LIN {X 0,Y 424.138,Z 935.188,A -85,B 0,C 180,E1 -9807.151,E2 -9807.151} C_VEL
LIN {X 0,Y 424.125,Z 936.443,A -85,B 0,C 180,E1 -9808.101,E2 -9808.101} C_VEL
LIN {X 0,Y 424.085,Z 937.224,A -85,B 0,C 180,E1 -9809.05,E2 -9809.05} C_VEL
LIN {X 0,Y 424.081,Z 937.52,A -85,B 0,C 180,E1 -9810,E2 -9810} C_VEL
LIN {X 0,Y 424.085,Z 937.223,A -85,B 0,C 180,E1 -9810.95,E2 -9810.95} C_VEL
LIN {X 0,Y 424.125,Z 936.441,A -85,B 0,C 180,E1 -9811.899,E2 -9811.899} C_VEL
LIN {X 0,Y 424.138,Z 935.183,A -85,B 0,C 180,E1 -9812.849,E2 -9812.849} C_VEL
LIN {X 0,Y 424.185,Z 932.271,A -85,B 0,C 180,E1 -9814.276,E2 -9814.276} C_VEL
LIN {X 0,Y 424.292,Z 929.619,A -85,B 0,C 180,E1 -9815.227,E2 -9815.227} C_VEL
LIN {X 0,Y 424.459,Z 924.427,A -85,B 0,C 180,E1 -9816.656,E2 -9816.656} C_VEL
LIN {X 0,Y 424.787,Z 917.59,A -85,B 0,C 180,E1 -9818.084,E2 -9818.084} C_VEL
LIN {X 0,Y 425.186,Z 910.116,A -85,B 0,C 180,E1 -9819.274,E2 -9819.274} C_VEL
LIN {X 0,Y 425.577,Z 902.747,A -85,B 0,C 180,E1 -9820.226,E2 -9820.226} C_VEL
LIN {X 0,Y 426.04,Z 894.86,A -85,B 0,C 180,E1 -9821.056,E2 -9821.056} C_VEL
LIN {X 0,Y 426.464,Z 886.526,A -85,B 0,C 180,E1 -9821.767,E2 -9821.767} C_VEL
LIN {X 0,Y 426.955,Z 877.803,A -85,B 0,C 180,E1 -9822.356,E2 -9822.356} C_VEL
LIN {X 0,Y 427.276,Z 865.987,A -85,B 0,C 180,E1 -9822.951,E2 -9822.951} C_VEL
LIN {X 0,Y 427.656,Z 855.955,A -85,B 0,C 180,E1 -9823.271,E2 -9823.271} C_VEL
LIN {X 0,Y 427.862,Z 833.743,A -85,B 0,C 180,E1 -9823.678,E2 -9823.678} C_VEL
LIN {X 0,Y 427.935,Z 796.078,A -85,B 0,C 180,E1 -9824.313,E2 -9824.313} C_VEL
LIN {X 0,Y 425.44,Z 777.594,A -85,B 0,C 180,E1 -9824.737,E2 -9824.737} C_VEL
LIN {X 0,Y 425.535,Z 774.648,A -85,B 0,C 180,E1 -9825.322,E2 -9825.322} C_VEL
LIN {X 0,Y 426.176,Z 760.658,A -85,B 0,C 180,E1 -9828.509,E2 -9828.509} C_VEL
LIN {X 0,Y 427.088,Z 745.503,A -85,B 0,C 180,E1 -9831.985,E2 -9831.985} C_VEL
LIN {X 0,Y 426.388,Z 740.059,A -85,B 0,C 180,E1 -9833.302,E2 -9833.302} C_VEL
LIN {X 0,Y 425.384,Z 734.368,A -85,B 0,C 180,E1 -9834.762,E2 -9834.762} C_VEL
LIN {X 0,Y 425.35,Z 734.312,A -85,B 0,C 180,E1 -9837.558,E2 -9837.558} C_VEL
LIN {X 0,Y 425.288,Z 734.304,A -85,B 0,C 180,E1 -9840.816,E2 -9840.816} C_VEL
LIN {X 0,Y 425.312,Z 734.317,A -85,B 0,C 180,E1 -9844.288,E2 -9844.288} C_VEL
LIN {X 0,Y 425.287,Z 734.323,A -85,B 0,C 180,E1 -9847.693,E2 -9847.693} C_VEL
LIN {X 0,Y 425.286,Z 734.31,A -85,B 0,C 180,E1 -9850.521,E2 -9850.521} C_VEL
LIN {X 0,Y 425.266,Z 734.324,A -85,B 0,C 180,E1 -9853.955,E2 -9853.955} C_VEL
LIN {X 0,Y 425.282,Z 734.317,A -85,B 0,C 180,E1 -9857.348,E2 -9857.348} C_VEL
LIN {X 0,Y 425.308,Z 734.283,A -85,B 0,C 180,E1 -9859.875,E2 -9859.875} C_VEL
LIN {X 0,Y 425.287,Z 734.303,A -85,B 0,C 180,E1 -9862.487,E2 -9862.487} C_VEL
LIN {X 0,Y 425.309,Z 734.32,A -85,B 0,C 180,E1 -9865.818,E2 -9865.818} C_VEL
LIN {X 0,Y 425.291,Z 734.315,A -85,B 0,C 180,E1 -9869.239,E2 -9869.239} C_VEL
LIN {X 0,Y 425.351,Z 734.311,A -85,B 0,C 180,E1 -9872.443,E2 -9872.443} C_VEL
LIN {X 0,Y 425.353,Z 734.312,A -85,B 0,C 180,E1 -9875.602,E2 -9875.602} C_VEL
LIN {X 0,Y 425.295,Z 734.306,A -85,B 0,C 180,E1 -9878.682,E2 -9878.682} C_VEL
LIN {X 0,Y 425.335,Z 734.311,A -85,B 0,C 180,E1 -9881.703,E2 -9881.703} C_VEL
LIN {X 0,Y 425.35,Z 734.308,A -85,B 0,C 180,E1 -9884.671,E2 -9884.671} C_VEL
LIN {X 0,Y 425.414,Z 734.289,A -85,B 0,C 180,E1 -9887.598,E2 -9887.598} C_VEL
LIN {X 0,Y 425.444,Z 734.297,A -85,B 0,C 180,E1 -9891.45,E2 -9891.45} C_VEL
LIN {X 0,Y 425.553,Z 734.289,A -85,B 0,C 180,E1 -9894.313,E2 -9894.313} C_VEL
LIN {X 0,Y 425.575,Z 734.267,A -85,B 0,C 180,E1 -9898.107,E2 -9898.107} C_VEL
LIN {X 0,Y 425.706,Z 734.26,A -85,B 0,C 180,E1 -9900,E2 -9900} C_VEL
LIN {X 0,Y 425.559,Z 734.287,A -85,B 0,C 180,E1 -9902.84,E2 -9902.84} C_VEL
LIN {X 0,Y 425.53,Z 734.277,A -85,B 0,C 180,E1 -9906.639,E2 -9906.639} C_VEL
LIN {X 0,Y 425.402,Z 734.298,A -85,B 0,C 180,E1 -9909.509,E2 -9909.509} C_VEL
LIN {X 0,Y 425.395,Z 734.31,A -85,B 0,C 180,E1 -9912.904,E2 -9912.904} C_VEL
LIN {X 0,Y 425.363,Z 734.301,A -85,B 0,C 180,E1 -9916.605,E2 -9916.605} C_VEL
LIN {X 0,Y 425.33,Z 734.31,A -85,B 0,C 180,E1 -9919.636,E2 -9919.636} C_VEL
LIN {X 0,Y 425.289,Z 734.319,A -85,B 0,C 180,E1 -9922.339,E2 -9922.339} C_VEL
LIN {X 0,Y 425.293,Z 734.307,A -85,B 0,C 180,E1 -9925.446,E2 -9925.446} C_VEL
LIN {X 0,Y 425.35,Z 734.31,A -85,B 0,C 180,E1 -9927.558,E2 -9927.558} C_VEL
LIN {X 0,Y 425.289,Z 734.321,A -85,B 0,C 180,E1 -9930.816,E2 -9930.816} C_VEL
LIN {X 0,Y 425.311,Z 734.309,A -85,B 0,C 180,E1 -9934.288,E2 -9934.288} C_VEL
LIN {X 0,Y 425.28,Z 734.32,A -85,B 0,C 180,E1 -9937.694,E2 -9937.694} C_VEL
LIN {X 0,Y 425.278,Z 734.308,A -85,B 0,C 180,E1 -9940.52,E2 -9940.52} C_VEL
LIN {X 0,Y 425.262,Z 734.307,A -85,B 0,C 180,E1 -9943.956,E2 -9943.956} C_VEL
LIN {X 0,Y 425.275,Z 734.325,A -85,B 0,C 180,E1 -9947.347,E2 -9947.347} C_VEL
LIN {X 0,Y 425.286,Z 734.312,A -85,B 0,C 180,E1 -9949.873,E2 -9949.873} C_VEL
LIN {X 0,Y 425.278,Z 734.311,A -85,B 0,C 180,E1 -9952.489,E2 -9952.489} C_VEL
LIN {X 0,Y 425.307,Z 734.321,A -85,B 0,C 180,E1 -9955.817,E2 -9955.817} C_VEL
LIN {X 0,Y 425.291,Z 734.312,A -85,B 0,C 180,E1 -9959.239,E2 -9959.239} C_VEL
LIN {X 0,Y 425.273,Z 734.322,A -85,B 0,C 180,E1 -9962.437,E2 -9962.437} C_VEL
LIN {X 0,Y 425.347,Z 734.317,A -85,B 0,C 180,E1 -9965.602,E2 -9965.602} C_VEL
LIN {X 0,Y 425.3,Z 734.318,A -85,B 0,C 180,E1 -9968.682,E2 -9968.682} C_VEL
LIN {X 0,Y 425.396,Z 734.425,A -85,B 0,C 180,E1 -9969.783,E2 -9969.783} C_VEL
LIN {X 0,Y 426.02,Z 739.289,A -85,B 0,C 180,E1 -9971.235,E2 -9971.235} C_VEL
LIN {X 0,Y 425.751,Z 748.087,A -85,B 0,C 180,E1 -9973.703,E2 -9973.703} C_VEL
LIN {X 0,Y 425.491,Z 754.134,A -85,B 0,C 180,E1 -9975.297,E2 -9975.297} C_VEL
LIN {X 0,Y 426.166,Z 757.896,A -85,B 0,C 180,E1 -9975.435,E2 -9975.435} C_VEL
LIN {X 0,Y 428.26,Z 770.133,A -85,B 0,C 180,E1 -9975.717,E2 -9975.717} C_VEL
LIN {X 0,Y 427.782,Z 829.524,A -85,B 0,C 180,E1 -9976.733,E2 -9976.733} C_VEL
LIN {X 0,Y 427.629,Z 839.402,A -85,B 0,C 180,E1 -9977.03,E2 -9977.03} C_VEL
LIN {X 0,Y 427.198,Z 850.542,A -85,B 0,C 180,E1 -9977.53,E2 -9977.53} C_VEL
LIN {X 0,Y 426.816,Z 861.387,A -85,B 0,C 180,E1 -9978.243,E2 -9978.243} C_VEL
LIN {X 0,Y 426.333,Z 869.786,A -85,B 0,C 180,E1 -9978.952,E2 -9978.952} C_VEL
LIN {X 0,Y 425.93,Z 877.709,A -85,B 0,C 180,E1 -9979.783,E2 -9979.783} C_VEL
LIN {X 0,Y 425.588,Z 883.399,A -85,B 0,C 180,E1 -9980.495,E2 -9980.495} C_VEL
LIN {X 0,Y 425.435,Z 885.864,A -85,B 0,C 180,E1 -9980.84,E2 -9980.84} C_VEL
LIN {X 0,Y 424.575,Z 889.849,A -85,B 0,C 180,E1 -9981.419,E2 -9981.419} C_VEL
LIN {X 0,Y 421.471,Z 895.791,A -85,B 0,C 180,E1 -9982.412,E2 -9982.412} C_VEL
LIN {X 0,Y 418.358,Z 900.822,A -85,B 0,C 180,E1 -9983.502,E2 -9983.502} C_VEL
LIN {X 0,Y 417.496,Z 903.376,A -85,B 0,C 180,E1 -9984.225,E2 -9984.225} C_VEL
LIN {X 0,Y 417.271,Z 906.303,A -85,B 0,C 180,E1 -9985.169,E2 -9985.169} C_VEL
LIN {X 0,Y 417.217,Z 908.62,A -85,B 0,C 180,E1 -9986.136,E2 -9986.136} C_VEL
LIN {X 0,Y 417.187,Z 910.384,A -85,B 0,C 180,E1 -9987.103,E2 -9987.103} C_VEL
LIN {X 0,Y 417.082,Z 911.659,A -85,B 0,C 180,E1 -9988.069,E2 -9988.069} C_VEL
LIN {X 0,Y 417.012,Z 912.464,A -85,B 0,C 180,E1 -9989.034,E2 -9989.034} C_VEL
LIN {X 0,Y 417.002,Z 912.77,A -85,B 0,C 180,E1 -9990,E2 -9990} C_VEL
LIN {X 0,Y 417.012,Z 912.495,A -85,B 0,C 180,E1 -9990.966,E2 -9990.966} C_VEL
LIN {X 0,Y 417.082,Z 911.751,A -85,B 0,C 180,E1 -9991.931,E2 -9991.931} C_VEL
LIN {X 0,Y 417.186,Z 910.54,A -85,B 0,C 180,E1 -9992.897,E2 -9992.897} C_VEL
LIN {X 0,Y 417.249,Z 907.697,A -85,B 0,C 180,E1 -9994.347,E2 -9994.347} C_VEL
LIN {X 0,Y 417.362,Z 905.108,A -85,B 0,C 180,E1 -9995.314,E2 -9995.314} C_VEL
LIN {X 0,Y 417.689,Z 900.007,A -85,B 0,C 180,E1 -9996.764,E2 -9996.764} C_VEL
LIN {X 0,Y 417.909,Z 894.523,A -85,B 0,C 180,E1 -9997.975,E2 -9997.975} C_VEL
LIN {X 0,Y 418.366,Z 887.629,A -85,B 0,C 180,E1 -9999.183,E2 -9999.183} C_VEL
LIN {X 0,Y 418.886,Z 879.709,A -85,B 0,C 180,E1 -10000.269,E2 -10000.269} C_VEL
LIN {X 0,Y 419.285,Z 872.158,A -85,B 0,C 180,E1 -10001.114,E2 -10001.114} C_VEL
LIN {X 0,Y 419.706,Z 864.241,A -85,B 0,C 180,E1 -10001.837,E2 -10001.837} C_VEL
LIN {X 0,Y 420.074,Z 856.064,A -85,B 0,C 180,E1 -10002.439,E2 -10002.439} C_VEL
LIN {X 0,Y 420.485,Z 847.776,A -85,B 0,C 180,E1 -10002.918,E2 -10002.918} C_VEL
LIN {X 0,Y 420.763,Z 838.827,A -85,B 0,C 180,E1 -10003.308,E2 -10003.308} C_VEL
LIN {X 0,Y 420.914,Z 829.602,A -85,B 0,C 180,E1 -10003.585,E2 -10003.585} C_VEL
LIN {X 0,Y 421.274,Z 770.019,A -85,B 0,C 180,E1 -10004.625,E2 -10004.625} C_VEL
LIN {X 0,Y 418.456,Z 754.177,A -85,B 0,C 180,E1 -10005.027,E2 -10005.027} C_VEL
LIN {X 0,Y 418.992,Z 743.301,A -85,B 0,C 180,E1 -10008.078,E2 -10008.078} C_VEL
LIN {X 0,Y 418.819,Z 738.045,A -85,B 0,C 180,E1 -10009.61,E2 -10009.61} C_VEL
LIN {X 0,Y 418.337,Z 735.274,A -85,B 0,C 180,E1 -10010.501,E2 -10010.501} C_VEL
LIN {X 0,Y 418.274,Z 735.191,A -85,B 0,C 180,E1 -10013.782,E2 -10013.782} C_VEL
LIN {X 0,Y 418.226,Z 735.2,A -85,B 0,C 180,E1 -10017.047,E2 -10017.047} C_VEL
LIN {X 0,Y 418.243,Z 735.198,A -85,B 0,C 180,E1 -10020.272,E2 -10020.272} C_VEL
LIN {X 0,Y 418.249,Z 735.195,A -85,B 0,C 180,E1 -10023.677,E2 -10023.677} C_VEL
LIN {X 0,Y 418.24,Z 735.188,A -85,B 0,C 180,E1 -10027.224,E2 -10027.224} C_VEL
LIN {X 0,Y 418.244,Z 735.185,A -85,B 0,C 180,E1 -10029.683,E2 -10029.683} C_VEL
LIN {X 0,Y 418.231,Z 735.201,A -85,B 0,C 180,E1 -10032.321,E2 -10032.321} C_VEL
LIN {X 0,Y 418.237,Z 735.187,A -85,B 0,C 180,E1 -10035.109,E2 -10035.109} C_VEL
LIN {X 0,Y 418.235,Z 735.163,A -85,B 0,C 180,E1 -10037.766,E2 -10037.766} C_VEL
LIN {X 0,Y 418.25,Z 735.188,A -85,B 0,C 180,E1 -10040.62,E2 -10040.62} C_VEL
LIN {X 0,Y 418.244,Z 735.196,A -85,B 0,C 180,E1 -10043.976,E2 -10043.976} C_VEL
LIN {X 0,Y 418.258,Z 735.191,A -85,B 0,C 180,E1 -10047.156,E2 -10047.156} C_VEL
LIN {X 0,Y 418.27,Z 735.199,A -85,B 0,C 180,E1 -10050.895,E2 -10050.895} C_VEL
LIN {X 0,Y 418.27,Z 735.179,A -85,B 0,C 180,E1 -10054.096,E2 -10054.096} C_VEL
LIN {X 0,Y 418.234,Z 735.202,A -85,B 0,C 180,E1 -10057.263,E2 -10057.263} C_VEL
LIN {X 0,Y 418.285,Z 735.188,A -85,B 0,C 180,E1 -10060.364,E2 -10060.364} C_VEL
LIN {X 0,Y 418.318,Z 735.178,A -85,B 0,C 180,E1 -10063.405,E2 -10063.405} C_VEL
LIN {X 0,Y 418.348,Z 735.185,A -85,B 0,C 180,E1 -10066.999,E2 -10066.999} C_VEL
LIN {X 0,Y 418.342,Z 735.177,A -85,B 0,C 180,E1 -10070.329,E2 -10070.329} C_VEL
LIN {X 0,Y 418.515,Z 735.143,A -85,B 0,C 180,E1 -10072.279,E2 -10072.279} C_VEL
LIN {X 0,Y 418.513,Z 735.155,A -85,B 0,C 180,E1 -10074.217,E2 -10074.217} C_VEL
LIN {X 0,Y 418.547,Z 735.157,A -85,B 0,C 180,E1 -10078.075,E2 -10078.075} C_VEL
LIN {X 0,Y 418.673,Z 735.136,A -85,B 0,C 180,E1 -10080,E2 -10080} C_VEL
LIN {X 0,Y 418.503,Z 735.146,A -85,B 0,C 180,E1 -10082.888,E2 -10082.888} C_VEL
LIN {X 0,Y 418.49,Z 735.164,A -85,B 0,C 180,E1 -10086.751,E2 -10086.751} C_VEL
LIN {X 0,Y 418.343,Z 735.183,A -85,B 0,C 180,E1 -10089.671,E2 -10089.671} C_VEL
LIN {X 0,Y 418.348,Z 735.168,A -85,B 0,C 180,E1 -10093.001,E2 -10093.001} C_VEL
LIN {X 0,Y 418.315,Z 735.186,A -85,B 0,C 180,E1 -10096.736,E2 -10096.736} C_VEL
LIN {X 0,Y 418.301,Z 735.185,A -85,B 0,C 180,E1 -10099.801,E2 -10099.801} C_VEL
LIN {X 0,Y 418.29,Z 735.189,A -85,B 0,C 180,E1 -10103.781,E2 -10103.781} C_VEL
LIN {X 0,Y 418.311,Z 735.185,A -85,B 0,C 180,E1 -10107.07,E2 -10107.07} C_VEL
LIN {X 0,Y 418.245,Z 735.192,A -85,B 0,C 180,E1 -10110.272,E2 -10110.272} C_VEL
LIN {X 0,Y 418.25,Z 735.197,A -85,B 0,C 180,E1 -10113.677,E2 -10113.677} C_VEL
LIN {X 0,Y 418.248,Z 735.178,A -85,B 0,C 180,E1 -10117.223,E2 -10117.223} C_VEL
LIN {X 0,Y 418.264,Z 735.157,A -85,B 0,C 180,E1 -10119.68,E2 -10119.68} C_VEL
LIN {X 0,Y 418.246,Z 735.188,A -85,B 0,C 180,E1 -10122.323,E2 -10122.323} C_VEL
LIN {X 0,Y 418.238,Z 735.197,A -85,B 0,C 180,E1 -10125.109,E2 -10125.109} C_VEL
LIN {X 0,Y 418.241,Z 735.188,A -85,B 0,C 180,E1 -10127.767,E2 -10127.767} C_VEL
LIN {X 0,Y 418.262,Z 735.195,A -85,B 0,C 180,E1 -10130.618,E2 -10130.618} C_VEL
LIN {X 0,Y 418.247,Z 735.191,A -85,B 0,C 180,E1 -10133.976,E2 -10133.976} C_VEL
LIN {X 0,Y 418.258,Z 735.193,A -85,B 0,C 180,E1 -10137.156,E2 -10137.156} C_VEL
LIN {X 0,Y 418.269,Z 735.192,A -85,B 0,C 180,E1 -10140.895,E2 -10140.895} C_VEL
LIN {X 0,Y 418.284,Z 735.187,A -85,B 0,C 180,E1 -10144.097,E2 -10144.097} C_VEL
LIN {X 0,Y 418.359,Z 735.384,A -85,B 0,C 180,E1 -10145.113,E2 -10145.113} C_VEL
LIN {X 0,Y 420.069,Z 745.334,A -85,B 0,C 180,E1 -10147.628,E2 -10147.628} C_VEL
LIN {X 0,Y 419.508,Z 755.719,A -85,B 0,C 180,E1 -10150.063,E2 -10150.063} C_VEL
LIN {X 0,Y 418.7,Z 770.161,A -85,B 0,C 180,E1 -10153.42,E2 -10153.42} C_VEL
LIN {X 0,Y 418.41,Z 777.042,A -85,B 0,C 180,E1 -10154.972,E2 -10154.972} C_VEL
LIN {X 0,Y 418.872,Z 780.553,A -85,B 0,C 180,E1 -10155.103,E2 -10155.103} C_VEL
LIN {X 0,Y 421.207,Z 799.105,A -85,B 0,C 180,E1 -10155.506,E2 -10155.506} C_VEL
LIN {X 0,Y 420.834,Z 853.261,A -85,B 0,C 180,E1 -10156.448,E2 -10156.448} C_VEL
LIN {X 0,Y 420.538,Z 862.53,A -85,B 0,C 180,E1 -10156.715,E2 -10156.715} C_VEL
LIN {X 0,Y 420.215,Z 871,A -85,B 0,C 180,E1 -10157.074,E2 -10157.074} C_VEL
LIN {X 0,Y 419.87,Z 879.511,A -85,B 0,C 180,E1 -10157.555,E2 -10157.555} C_VEL
LIN {X 0,Y 419.437,Z 887.855,A -85,B 0,C 180,E1 -10158.155,E2 -10158.155} C_VEL
LIN {X 0,Y 418.989,Z 895.908,A -85,B 0,C 180,E1 -10158.878,E2 -10158.878} C_VEL
LIN {X 0,Y 418.501,Z 904.603,A -85,B 0,C 180,E1 -10159.844,E2 -10159.844} C_VEL
LIN {X 0,Y 417.969,Z 913.134,A -85,B 0,C 180,E1 -10161.052,E2 -10161.052} C_VEL
LIN {X 0,Y 417.609,Z 919.832,A -85,B 0,C 180,E1 -10162.263,E2 -10162.263} C_VEL
LIN {X 0,Y 417.342,Z 925.259,A -85,B 0,C 180,E1 -10163.491,E2 -10163.491} C_VEL
LIN {X 0,Y 417.21,Z 929.418,A -85,B 0,C 180,E1 -10164.684,E2 -10164.684} C_VEL
LIN {X 0,Y 417.11,Z 932.069,A -85,B 0,C 180,E1 -10165.652,E2 -10165.652} C_VEL
LIN {X 0,Y 417.037,Z 934.979,A -85,B 0,C 180,E1 -10167.102,E2 -10167.102} C_VEL
LIN {X 0,Y 417.053,Z 936.236,A -85,B 0,C 180,E1 -10168.069,E2 -10168.069} C_VEL
LIN {X 0,Y 417.008,Z 937.016,A -85,B 0,C 180,E1 -10169.034,E2 -10169.034} C_VEL
LIN {X 0,Y 417.001,Z 937.312,A -85,B 0,C 180,E1 -10170,E2 -10170} C_VEL
LIN {X 0,Y 417.008,Z 937.015,A -85,B 0,C 180,E1 -10170.966,E2 -10170.966} C_VEL
LIN {X 0,Y 417.053,Z 936.232,A -85,B 0,C 180,E1 -10171.931,E2 -10171.931} C_VEL
LIN {X 0,Y 417.037,Z 934.974,A -85,B 0,C 180,E1 -10172.898,E2 -10172.898} C_VEL
LIN {X 0,Y 417.11,Z 932.062,A -85,B 0,C 180,E1 -10174.348,E2 -10174.348} C_VEL
LIN {X 0,Y 417.21,Z 929.409,A -85,B 0,C 180,E1 -10175.316,E2 -10175.316} C_VEL
LIN {X 0,Y 417.342,Z 925.247,A -85,B 0,C 180,E1 -10176.509,E2 -10176.509} C_VEL
LIN {X 0,Y 417.609,Z 919.813,A -85,B 0,C 180,E1 -10177.737,E2 -10177.737} C_VEL
LIN {X 0,Y 417.965,Z 913.117,A -85,B 0,C 180,E1 -10178.948,E2 -10178.948} C_VEL
LIN {X 0,Y 418.5,Z 904.585,A -85,B 0,C 180,E1 -10180.156,E2 -10180.156} C_VEL
LIN {X 0,Y 418.954,Z 897.115,A -85,B 0,C 180,E1 -10181,E2 -10181} C_VEL
LIN {X 0,Y 419.373,Z 889.321,A -85,B 0,C 180,E1 -10181.724,E2 -10181.724} C_VEL
LIN {X 0,Y 419.796,Z 881.339,A -85,B 0,C 180,E1 -10182.325,E2 -10182.325} C_VEL
LIN {X 0,Y 420.189,Z 872.15,A -85,B 0,C 180,E1 -10182.865,E2 -10182.865} C_VEL
LIN {X 0,Y 420.483,Z 863.274,A -85,B 0,C 180,E1 -10183.256,E2 -10183.256} C_VEL
LIN {X 0,Y 420.799,Z 854.437,A -85,B 0,C 180,E1 -10183.522,E2 -10183.522} C_VEL
LIN {X 0,Y 421.202,Z 797.961,A -85,B 0,C 180,E1 -10184.511,E2 -10184.511} C_VEL
LIN {X 0,Y 418.447,Z 777.572,A -85,B 0,C 180,E1 -10184.977,E2 -10184.977} C_VEL
LIN {X 0,Y 418.463,Z 775.625,A -85,B 0,C 180,E1 -10185.313,E2 -10185.313} C_VEL
LIN {X 0,Y 419.151,Z 761.55,A -85,B 0,C 180,E1 -10188.577,E2 -10188.577} C_VEL
LIN {X 0,Y 420.041,Z 747.487,A -85,B 0,C 180,E1 -10191.856,E2 -10191.856} C_VEL
LIN {X 0,Y 419.966,Z 744.236,A -85,B 0,C 180,E1 -10192.637,E2 -10192.637} C_VEL
LIN {X 0,Y 418.322,Z 735.236,A -85,B 0,C 180,E1 -10194.955,E2 -10194.955} C_VEL
LIN {X 0,Y 418.292,Z 735.194,A -85,B 0,C 180,E1 -10198.063,E2 -10198.063} C_VEL
LIN {X 0,Y 418.212,Z 735.188,A -85,B 0,C 180,E1 -10201.396,E2 -10201.396} C_VEL
LIN {X 0,Y 418.266,Z 735.195,A -85,B 0,C 180,E1 -10204.58,E2 -10204.58} C_VEL
LIN {X 0,Y 418.236,Z 735.2,A -85,B 0,C 180,E1 -10207.835,E2 -10207.835} C_VEL
LIN {X 0,Y 418.224,Z 735.189,A -85,B 0,C 180,E1 -10210.948,E2 -10210.948} C_VEL
LIN {X 0,Y 418.215,Z 735.203,A -85,B 0,C 180,E1 -10213.73,E2 -10213.73} C_VEL
LIN {X 0,Y 418.209,Z 735.197,A -85,B 0,C 180,E1 -10216.449,E2 -10216.449} C_VEL
LIN {X 0,Y 418.266,Z 735.174,A -85,B 0,C 180,E1 -10219.124,E2 -10219.124} C_VEL
LIN {X 0,Y 418.238,Z 735.177,A -85,B 0,C 180,E1 -10222.165,E2 -10222.165} C_VEL
LIN {X 0,Y 418.267,Z 735.192,A -85,B 0,C 180,E1 -10225.42,E2 -10225.42} C_VEL
LIN {X 0,Y 418.212,Z 735.196,A -85,B 0,C 180,E1 -10228.604,E2 -10228.604} C_VEL
LIN {X 0,Y 418.293,Z 735.187,A -85,B 0,C 180,E1 -10231.937,E2 -10231.937} C_VEL
LIN {X 0,Y 418.291,Z 735.189,A -85,B 0,C 180,E1 -10235.163,E2 -10235.163} C_VEL
LIN {X 0,Y 418.235,Z 735.186,A -85,B 0,C 180,E1 -10238.304,E2 -10238.304} C_VEL
LIN {X 0,Y 418.286,Z 735.187,A -85,B 0,C 180,E1 -10241.383,E2 -10241.383} C_VEL
LIN {X 0,Y 418.304,Z 735.189,A -85,B 0,C 180,E1 -10244.406,E2 -10244.406} C_VEL
LIN {X 0,Y 418.357,Z 735.166,A -85,B 0,C 180,E1 -10247.386,E2 -10247.386} C_VEL
LIN {X 0,Y 418.343,Z 735.183,A -85,B 0,C 180,E1 -10250.329,E2 -10250.329} C_VEL
LIN {X 0,Y 418.49,Z 735.164,A -85,B 0,C 180,E1 -10253.249,E2 -10253.249} C_VEL
LIN {X 0,Y 418.341,Z 735.177,A -85,B 0,C 180,E1 -10255.182,E2 -10255.182} C_VEL
LIN {X 0,Y 418.545,Z 735.142,A -85,B 0,C 180,E1 -10258.076,E2 -10258.076} C_VEL
LIN {X 0,Y 418.675,Z 735.135,A -85,B 0,C 180,E1 -10260,E2 -10260} C_VEL
LIN {X 0,Y 418.513,Z 735.164,A -85,B 0,C 180,E1 -10262.888,E2 -10262.888} C_VEL
LIN {X 0,Y 418.493,Z 735.152,A -85,B 0,C 180,E1 -10266.751,E2 -10266.751} C_VEL
LIN {X 0,Y 418.402,Z 735.165,A -85,B 0,C 180,E1 -10268.695,E2 -10268.695} C_VEL
LIN {X 0,Y 418.317,Z 735.186,A -85,B 0,C 180,E1 -10271.631,E2 -10271.631} C_VEL
LIN {X 0,Y 418.305,Z 735.191,A -85,B 0,C 180,E1 -10274.597,E2 -10274.597} C_VEL
LIN {X 0,Y 418.282,Z 735.179,A -85,B 0,C 180,E1 -10277.604,E2 -10277.604} C_VEL
LIN {X 0,Y 418.252,Z 735.196,A -85,B 0,C 180,E1 -10280.663,E2 -10280.663} C_VEL
LIN {X 0,Y 418.277,Z 735.187,A -85,B 0,C 180,E1 -10283.782,E2 -10283.782} C_VEL
LIN {X 0,Y 418.312,Z 735.182,A -85,B 0,C 180,E1 -10287.071,E2 -10287.071} C_VEL
LIN {X 0,Y 418.246,Z 735.195,A -85,B 0,C 180,E1 -10290.272,E2 -10290.272} C_VEL
LIN {X 0,Y 418.248,Z 735.19,A -85,B 0,C 180,E1 -10293.677,E2 -10293.677} C_VEL
LIN {X 0,Y 418.241,Z 735.203,A -85,B 0,C 180,E1 -10297.224,E2 -10297.224} C_VEL
LIN {X 0,Y 418.247,Z 735.186,A -85,B 0,C 180,E1 -10299.683,E2 -10299.683} C_VEL
LIN {X 0,Y 418.225,Z 735.163,A -85,B 0,C 180,E1 -10302.32,E2 -10302.32} C_VEL
LIN {X 0,Y 418.237,Z 735.187,A -85,B 0,C 180,E1 -10305.109,E2 -10305.109} C_VEL
LIN {X 0,Y 418.241,Z 735.2,A -85,B 0,C 180,E1 -10307.767,E2 -10307.767} C_VEL
LIN {X 0,Y 418.246,Z 735.185,A -85,B 0,C 180,E1 -10310.621,E2 -10310.621} C_VEL
LIN {X 0,Y 418.244,Z 735.201,A -85,B 0,C 180,E1 -10313.976,E2 -10313.976} C_VEL
LIN {X 0,Y 418.258,Z 735.195,A -85,B 0,C 180,E1 -10317.156,E2 -10317.156} C_VEL
LIN {X 0,Y 418.262,Z 735.194,A -85,B 0,C 180,E1 -10320.838,E2 -10320.838} C_VEL
LIN {X 0,Y 418.238,Z 735.2,A -85,B 0,C 180,E1 -10324.094,E2 -10324.094} C_VEL
LIN {X 0,Y 418.233,Z 735.197,A -85,B 0,C 180,E1 -10327.264,E2 -10327.264} C_VEL
LIN {X 0,Y 418.369,Z 735.38,A -85,B 0,C 180,E1 -10329.67,E2 -10329.67} C_VEL
LIN {X 0,Y 419.046,Z 741.219,A -85,B 0,C 180,E1 -10331.418,E2 -10331.418} C_VEL
LIN {X 0,Y 418.576,Z 751.831,A -85,B 0,C 180,E1 -10334.416,E2 -10334.416} C_VEL
LIN {X 0,Y 418.519,Z 754.337,A -85,B 0,C 180,E1 -10335.047,E2 -10335.047} C_VEL
LIN {X 0,Y 419.226,Z 758.605,A -85,B 0,C 180,E1 -10335.197,E2 -10335.197} C_VEL
LIN {X 0,Y 421.398,Z 770.767,A -85,B 0,C 180,E1 -10335.486,E2 -10335.486} C_VEL
LIN {X 0,Y 420.897,Z 829.753,A -85,B 0,C 180,E1 -10336.512,E2 -10336.512} C_VEL
LIN {X 0,Y 420.739,Z 839.623,A -85,B 0,C 180,E1 -10336.814,E2 -10336.814} C_VEL
LIN {X 0,Y 420.298,Z 850.759,A -85,B 0,C 180,E1 -10337.322,E2 -10337.322} C_VEL
LIN {X 0,Y 419.889,Z 861.601,A -85,B 0,C 180,E1 -10338.046,E2 -10338.046} C_VEL
LIN {X 0,Y 419.374,Z 869.999,A -85,B 0,C 180,E1 -10338.766,E2 -10338.766} C_VEL
LIN {X 0,Y 418.952,Z 877.921,A -85,B 0,C 180,E1 -10339.611,E2 -10339.611} C_VEL
LIN {X 0,Y 418.609,Z 883.611,A -85,B 0,C 180,E1 -10340.335,E2 -10340.335} C_VEL
LIN {X 0,Y 418.2,Z 889.96,A -85,B 0,C 180,E1 -10341.301,E2 -10341.301} C_VEL
LIN {X 0,Y 417.832,Z 896.405,A -85,B 0,C 180,E1 -10342.51,E2 -10342.51} C_VEL
LIN {X 0,Y 417.645,Z 901.542,A -85,B 0,C 180,E1 -10343.72,E2 -10343.72} C_VEL
LIN {X 0,Y 417.496,Z 903.376,A -85,B 0,C 180,E1 -10344.225,E2 -10344.225} C_VEL
LIN {X 0,Y 416.661,Z 905.75,A -85,B 0,C 180,E1 -10344.968,E2 -10344.968} C_VEL
LIN {X 0,Y 413.656,Z 908.943,A -85,B 0,C 180,E1 -10346.196,E2 -10346.196} C_VEL
LIN {X 0,Y 411.184,Z 910.836,A -85,B 0,C 180,E1 -10347.211,E2 -10347.211} C_VEL
LIN {X 0,Y 410.092,Z 911.841,A -85,B 0,C 180,E1 -10348.011,E2 -10348.011} C_VEL
LIN {X 0,Y 409.983,Z 912.071,A -85,B 0,C 180,E1 -10348.284,E2 -10348.284} C_VEL
LIN {X 0,Y 409.937,Z 912.672,A -85,B 0,C 180,E1 -10349.018,E2 -10349.018} C_VEL
LIN {X 0,Y 409.925,Z 912.979,A -85,B 0,C 180,E1 -10350,E2 -10350} C_VEL
LIN {X 0,Y 409.938,Z 912.703,A -85,B 0,C 180,E1 -10350.982,E2 -10350.982} C_VEL
LIN {X 0,Y 410.014,Z 911.959,A -85,B 0,C 180,E1 -10351.965,E2 -10351.965} C_VEL
LIN {X 0,Y 410.091,Z 910.748,A -85,B 0,C 180,E1 -10352.947,E2 -10352.947} C_VEL
LIN {X 0,Y 410.165,Z 907.905,A -85,B 0,C 180,E1 -10354.422,E2 -10354.422} C_VEL
LIN {X 0,Y 410.313,Z 905.315,A -85,B 0,C 180,E1 -10355.406,E2 -10355.406} C_VEL
LIN {X 0,Y 410.595,Z 901.364,A -85,B 0,C 180,E1 -10356.583,E2 -10356.583} C_VEL
LIN {X 0,Y 410.726,Z 897.181,A -85,B 0,C 180,E1 -10357.596,E2 -10357.596} C_VEL
LIN {X 0,Y 411.054,Z 892.124,A -85,B 0,C 180,E1 -10358.604,E2 -10358.604} C_VEL
LIN {X 0,Y 411.479,Z 886.159,A -85,B 0,C 180,E1 -10359.586,E2 -10359.586} C_VEL
LIN {X 0,Y 411.96,Z 878.897,A -85,B 0,C 180,E1 -10360.568,E2 -10360.568} C_VEL
LIN {X 0,Y 412.408,Z 871.135,A -85,B 0,C 180,E1 -10361.426,E2 -10361.426} C_VEL
LIN {X 0,Y 412.776,Z 864.443,A -85,B 0,C 180,E1 -10362.039,E2 -10362.039} C_VEL
LIN {X 0,Y 413.173,Z 856.265,A -85,B 0,C 180,E1 -10362.65,E2 -10362.65} C_VEL
LIN {X 0,Y 413.576,Z 847.976,A -85,B 0,C 180,E1 -10363.137,E2 -10363.137} C_VEL
LIN {X 0,Y 413.869,Z 839.023,A -85,B 0,C 180,E1 -10363.534,E2 -10363.534} C_VEL
LIN {X 0,Y 414.039,Z 829.883,A -85,B 0,C 180,E1 -10363.813,E2 -10363.813} C_VEL
LIN {X 0,Y 414.448,Z 771.134,A -85,B 0,C 180,E1 -10364.855,E2 -10364.855} C_VEL
LIN {X 0,Y 411.486,Z 754.375,A -85,B 0,C 180,E1 -10365.287,E2 -10365.287} C_VEL
LIN {X 0,Y 411.953,Z 745.249,A -85,B 0,C 180,E1 -10367.884,E2 -10367.884} C_VEL
LIN {X 0,Y 411.899,Z 739.977,A -85,B 0,C 180,E1 -10369.434,E2 -10369.434} C_VEL
LIN {X 0,Y 411.288,Z 736.163,A -85,B 0,C 180,E1 -10370.636,E2 -10370.636} C_VEL
LIN {X 0,Y 411.204,Z 736.075,A -85,B 0,C 180,E1 -10374.217,E2 -10374.217} C_VEL
LIN {X 0,Y 411.189,Z 736.076,A -85,B 0,C 180,E1 -10377.483,E2 -10377.483} C_VEL
LIN {X 0,Y 411.19,Z 736.069,A -85,B 0,C 180,E1 -10380.848,E2 -10380.848} C_VEL
LIN {X 0,Y 411.206,Z 736.078,A -85,B 0,C 180,E1 -10384.334,E2 -10384.334} C_VEL
LIN {X 0,Y 411.191,Z 736.063,A -85,B 0,C 180,E1 -10387.974,E2 -10387.974} C_VEL
LIN {X 0,Y 411.164,Z 736.078,A -85,B 0,C 180,E1 -10391.228,E2 -10391.228} C_VEL
LIN {X 0,Y 411.177,Z 736.074,A -85,B 0,C 180,E1 -10394.49,E2 -10394.49} C_VEL
LIN {X 0,Y 411.174,Z 736.044,A -85,B 0,C 180,E1 -10398.194,E2 -10398.194} C_VEL
LIN {X 0,Y 411.215,Z 736.066,A -85,B 0,C 180,E1 -10400.775,E2 -10400.775} C_VEL
LIN {X 0,Y 411.198,Z 736.077,A -85,B 0,C 180,E1 -10404.471,E2 -10404.471} C_VEL
LIN {X 0,Y 411.208,Z 736.067,A -85,B 0,C 180,E1 -10406.873,E2 -10406.873} C_VEL
LIN {X 0,Y 411.234,Z 736.073,A -85,B 0,C 180,E1 -10410.644,E2 -10410.644} C_VEL
LIN {X 0,Y 411.239,Z 736.056,A -85,B 0,C 180,E1 -10413.619,E2 -10413.619} C_VEL
LIN {X 0,Y 411.198,Z 736.073,A -85,B 0,C 180,E1 -10416.852,E2 -10416.852} C_VEL
LIN {X 0,Y 411.216,Z 736.068,A -85,B 0,C 180,E1 -10420.05,E2 -10420.05} C_VEL
LIN {X 0,Y 411.265,Z 736.054,A -85,B 0,C 180,E1 -10423.131,E2 -10423.131} C_VEL
LIN {X 0,Y 411.307,Z 736.061,A -85,B 0,C 180,E1 -10426.896,E2 -10426.896} C_VEL
LIN {X 0,Y 411.294,Z 736.055,A -85,B 0,C 180,E1 -10430.161,E2 -10430.161} C_VEL
LIN {X 0,Y 411.484,Z 736.018,A -85,B 0,C 180,E1 -10432.147,E2 -10432.147} C_VEL
LIN {X 0,Y 411.475,Z 736.032,A -85,B 0,C 180,E1 -10434.118,E2 -10434.118} C_VEL
LIN {X 0,Y 411.516,Z 736.034,A -85,B 0,C 180,E1 -10438.042,E2 -10438.042} C_VEL
LIN {X 0,Y 411.642,Z 736.011,A -85,B 0,C 180,E1 -10440,E2 -10440} C_VEL
LIN {X 0,Y 411.46,Z 736.023,A -85,B 0,C 180,E1 -10442.937,E2 -10442.937} C_VEL
LIN {X 0,Y 411.454,Z 736.041,A -85,B 0,C 180,E1 -10446.867,E2 -10446.867} C_VEL
LIN {X 0,Y 411.295,Z 736.058,A -85,B 0,C 180,E1 -10449.839,E2 -10449.839} C_VEL
LIN {X 0,Y 411.307,Z 736.045,A -85,B 0,C 180,E1 -10453.104,E2 -10453.104} C_VEL
LIN {X 0,Y 411.264,Z 736.065,A -85,B 0,C 180,E1 -10456.869,E2 -10456.869} C_VEL
LIN {X 0,Y 411.256,Z 736.059,A -85,B 0,C 180,E1 -10459.985,E2 -10459.985} C_VEL
LIN {X 0,Y 411.205,Z 736.066,A -85,B 0,C 180,E1 -10463.147,E2 -10463.147} C_VEL
LIN {X 0,Y 411.239,Z 736.07,A -85,B 0,C 180,E1 -10466.381,E2 -10466.381} C_VEL
LIN {X 0,Y 411.201,Z 736.064,A -85,B 0,C 180,E1 -10469.713,E2 -10469.713} C_VEL
LIN {X 0,Y 411.207,Z 736.072,A -85,B 0,C 180,E1 -10473.156,E2 -10473.156} C_VEL
LIN {X 0,Y 411.197,Z 736.06,A -85,B 0,C 180,E1 -10476.553,E2 -10476.553} C_VEL
LIN {X 0,Y 411.227,Z 736.032,A -85,B 0,C 180,E1 -10479.73,E2 -10479.73} C_VEL
LIN {X 0,Y 411.178,Z 736.074,A -85,B 0,C 180,E1 -10483.133,E2 -10483.133} C_VEL
LIN {X 0,Y 411.171,Z 736.078,A -85,B 0,C 180,E1 -10485.88,E2 -10485.88} C_VEL
LIN {X 0,Y 411.165,Z 736.067,A -85,B 0,C 180,E1 -10488.771,E2 -10488.771} C_VEL
LIN {X 0,Y 411.213,Z 736.073,A -85,B 0,C 180,E1 -10491.83,E2 -10491.83} C_VEL
LIN {X 0,Y 411.212,Z 736.075,A -85,B 0,C 180,E1 -10495.121,E2 -10495.121} C_VEL
LIN {X 0,Y 411.166,Z 736.073,A -85,B 0,C 180,E1 -10498.003,E2 -10498.003} C_VEL
LIN {X 0,Y 411.219,Z 736.075,A -85,B 0,C 180,E1 -10501.41,E2 -10501.41} C_VEL
LIN {X 0,Y 411.288,Z 736.122,A -85,B 0,C 180,E1 -10504.844,E2 -10504.844} C_VEL
LIN {X 0,Y 413.069,Z 746.242,A -85,B 0,C 180,E1 -10507.492,E2 -10507.492} C_VEL
LIN {X 0,Y 412.729,Z 752.74,A -85,B 0,C 180,E1 -10509.048,E2 -10509.048} C_VEL
LIN {X 0,Y 411.887,Z 767.632,A -85,B 0,C 180,E1 -10512.583,E2 -10512.583} C_VEL
LIN {X 0,Y 411.425,Z 776.841,A -85,B 0,C 180,E1 -10514.71,E2 -10514.71} C_VEL
LIN {X 0,Y 411.909,Z 780.794,A -85,B 0,C 180,E1 -10514.852,E2 -10514.852} C_VEL
LIN {X 0,Y 414.328,Z 798.914,A -85,B 0,C 180,E1 -10515.26,E2 -10515.26} C_VEL
LIN {X 0,Y 413.951,Z 853.121,A -85,B 0,C 180,E1 -10516.219,E2 -10516.219} C_VEL
LIN {X 0,Y 413.634,Z 862.33,A -85,B 0,C 180,E1 -10516.489,E2 -10516.489} C_VEL
LIN {X 0,Y 413.301,Z 870.797,A -85,B 0,C 180,E1 -10516.854,E2 -10516.854} C_VEL
LIN {X 0,Y 412.948,Z 879.307,A -85,B 0,C 180,E1 -10517.343,E2 -10517.343} C_VEL
LIN {X 0,Y 412.493,Z 887.65,A -85,B 0,C 180,E1 -10517.953,E2 -10517.953} C_VEL
LIN {X 0,Y 412.024,Z 895.702,A -85,B 0,C 180,E1 -10518.688,E2 -10518.688} C_VEL
LIN {X 0,Y 411.497,Z 904.396,A -85,B 0,C 180,E1 -10519.669,E2 -10519.669} C_VEL
LIN {X 0,Y 410.954,Z 912.927,A -85,B 0,C 180,E1 -10520.898,E2 -10520.898} C_VEL
LIN {X 0,Y 410.553,Z 919.624,A -85,B 0,C 180,E1 -10522.129,E2 -10522.129} C_VEL
LIN {X 0,Y 410.341,Z 924.023,A -85,B 0,C 180,E1 -10523.114,E2 -10523.114} C_VEL
LIN {X 0,Y 410.139,Z 927.682,A -85,B 0,C 180,E1 -10524.099,E2 -10524.099} C_VEL
LIN {X 0,Y 410.095,Z 930.689,A -85,B 0,C 180,E1 -10525.084,E2 -10525.084} C_VEL
LIN {X 0,Y 409.978,Z 933.018,A -85,B 0,C 180,E1 -10526.068,E2 -10526.068} C_VEL
LIN {X 0,Y 409.937,Z 934.77,A -85,B 0,C 180,E1 -10527.052,E2 -10527.052} C_VEL
LIN {X 0,Y 409.964,Z 936.027,A -85,B 0,C 180,E1 -10528.035,E2 -10528.035} C_VEL
LIN {X 0,Y 409.933,Z 936.808,A -85,B 0,C 180,E1 -10529.018,E2 -10529.018} C_VEL
LIN {X 0,Y 409.923,Z 937.104,A -85,B 0,C 180,E1 -10530,E2 -10530} C_VEL
LIN {X 0,Y 409.933,Z 936.807,A -85,B 0,C 180,E1 -10530.982,E2 -10530.982} C_VEL
LIN {X 0,Y 409.964,Z 936.023,A -85,B 0,C 180,E1 -10531.965,E2 -10531.965} C_VEL
LIN {X 0,Y 409.937,Z 934.764,A -85,B 0,C 180,E1 -10532.948,E2 -10532.948} C_VEL
LIN {X 0,Y 410.04,Z 931.853,A -85,B 0,C 180,E1 -10534.424,E2 -10534.424} C_VEL
LIN {X 0,Y 410.13,Z 929.199,A -85,B 0,C 180,E1 -10535.408,E2 -10535.408} C_VEL
LIN {X 0,Y 410.236,Z 925.63,A -85,B 0,C 180,E1 -10536.47,E2 -10536.47} C_VEL
LIN {X 0,Y 410.49,Z 920.78,A -85,B 0,C 180,E1 -10537.625,E2 -10537.625} C_VEL
LIN {X 0,Y 410.753,Z 915.75,A -85,B 0,C 180,E1 -10538.61,E2 -10538.61} C_VEL
LIN {X 0,Y 411.153,Z 909.694,A -85,B 0,C 180,E1 -10539.594,E2 -10539.594} C_VEL
LIN {X 0,Y 411.589,Z 902.324,A -85,B 0,C 180,E1 -10540.577,E2 -10540.577} C_VEL
LIN {X 0,Y 412.102,Z 894.436,A -85,B 0,C 180,E1 -10541.435,E2 -10541.435} C_VEL
LIN {X 0,Y 412.569,Z 886.101,A -85,B 0,C 180,E1 -10542.17,E2 -10542.17} C_VEL
LIN {X 0,Y 413.185,Z 875.463,A -85,B 0,C 180,E1 -10542.9,E2 -10542.9} C_VEL
LIN {X 0,Y 413.512,Z 863.888,A -85,B 0,C 180,E1 -10543.452,E2 -10543.452} C_VEL
LIN {X 0,Y 413.91,Z 854.215,A -85,B 0,C 180,E1 -10543.752,E2 -10543.752} C_VEL
LIN {X 0,Y 414.324,Z 798.677,A -85,B 0,C 180,E1 -10544.74,E2 -10544.74} C_VEL
LIN {X 0,Y 411.452,Z 777.361,A -85,B 0,C 180,E1 -10545.238,E2 -10545.238} C_VEL
LIN {X 0,Y 411.461,Z 775.42,A -85,B 0,C 180,E1 -10545.581,E2 -10545.581} C_VEL
LIN {X 0,Y 412.209,Z 761.359,A -85,B 0,C 180,E1 -10548.902,E2 -10548.902} C_VEL
LIN {X 0,Y 413.121,Z 747.309,A -85,B 0,C 180,E1 -10552.242,E2 -10552.242} C_VEL
LIN {X 0,Y 411.946,Z 739.692,A -85,B 0,C 180,E1 -10554.17,E2 -10554.17} C_VEL
LIN {X 0,Y 411.286,Z 736.09,A -85,B 0,C 180,E1 -10555.175,E2 -10555.175} C_VEL
LIN {X 0,Y 411.219,Z 736.075,A -85,B 0,C 180,E1 -10558.59,E2 -10558.59} C_VEL
LIN {X 0,Y 411.166,Z 736.075,A -85,B 0,C 180,E1 -10561.997,E2 -10561.997} C_VEL
LIN {X 0,Y 411.212,Z 736.075,A -85,B 0,C 180,E1 -10564.879,E2 -10564.879} C_VEL
LIN {X 0,Y 411.213,Z 736.073,A -85,B 0,C 180,E1 -10568.17,E2 -10568.17} C_VEL
LIN {X 0,Y 411.165,Z 736.067,A -85,B 0,C 180,E1 -10571.229,E2 -10571.229} C_VEL
LIN {X 0,Y 411.178,Z 736.076,A -85,B 0,C 180,E1 -10574.49,E2 -10574.49} C_VEL
LIN {X 0,Y 411.199,Z 736.058,A -85,B 0,C 180,E1 -10578.197,E2 -10578.197} C_VEL
LIN {X 0,Y 411.23,Z 736.029,A -85,B 0,C 180,E1 -10580.777,E2 -10580.777} C_VEL
LIN {X 0,Y 411.201,Z 736.07,A -85,B 0,C 180,E1 -10584.472,E2 -10584.472} C_VEL
LIN {X 0,Y 411.208,Z 736.072,A -85,B 0,C 180,E1 -10586.873,E2 -10586.873} C_VEL
LIN {X 0,Y 411.234,Z 736.059,A -85,B 0,C 180,E1 -10590.644,E2 -10590.644} C_VEL
LIN {X 0,Y 411.239,Z 736.07,A -85,B 0,C 180,E1 -10593.619,E2 -10593.619} C_VEL
LIN {X 0,Y 411.205,Z 736.066,A -85,B 0,C 180,E1 -10596.853,E2 -10596.853} C_VEL
LIN {X 0,Y 411.266,Z 736.058,A -85,B 0,C 180,E1 -10600.031,E2 -10600.031} C_VEL
LIN {X 0,Y 411.264,Z 736.065,A -85,B 0,C 180,E1 -10603.131,E2 -10603.131} C_VEL
LIN {X 0,Y 411.307,Z 736.045,A -85,B 0,C 180,E1 -10606.896,E2 -10606.896} C_VEL
LIN {X 0,Y 411.295,Z 736.058,A -85,B 0,C 180,E1 -10610.161,E2 -10610.161} C_VEL
LIN {X 0,Y 411.454,Z 736.041,A -85,B 0,C 180,E1 -10613.133,E2 -10613.133} C_VEL
LIN {X 0,Y 411.312,Z 736.053,A -85,B 0,C 180,E1 -10615.099,E2 -10615.099} C_VEL
LIN {X 0,Y 411.514,Z 736.017,A -85,B 0,C 180,E1 -10618.043,E2 -10618.043} C_VEL
LIN {X 0,Y 411.644,Z 736.011,A -85,B 0,C 180,E1 -10620,E2 -10620} C_VEL
LIN {X 0,Y 411.468,Z 736.041,A -85,B 0,C 180,E1 -10622.937,E2 -10622.937} C_VEL
LIN {X 0,Y 411.46,Z 736.025,A -85,B 0,C 180,E1 -10626.867,E2 -10626.867} C_VEL
LIN {X 0,Y 411.356,Z 736.045,A -85,B 0,C 180,E1 -10628.845,E2 -10628.845} C_VEL
LIN {X 0,Y 411.286,Z 736.062,A -85,B 0,C 180,E1 -10631.833,E2 -10631.833} C_VEL
LIN {X 0,Y 411.262,Z 736.064,A -85,B 0,C 180,E1 -10634.853,E2 -10634.853} C_VEL
LIN {X 0,Y 411.247,Z 736.054,A -85,B 0,C 180,E1 -10637.915,E2 -10637.915} C_VEL
LIN {X 0,Y 411.198,Z 736.08,A -85,B 0,C 180,E1 -10641.034,E2 -10641.034} C_VEL
LIN {X 0,Y 411.221,Z 736.066,A -85,B 0,C 180,E1 -10644.216,E2 -10644.216} C_VEL
LIN {X 0,Y 411.26,Z 736.065,A -85,B 0,C 180,E1 -10647.478,E2 -10647.478} C_VEL
LIN {X 0,Y 411.191,Z 736.078,A -85,B 0,C 180,E1 -10650.848,E2 -10650.848} C_VEL
LIN {X 0,Y 411.206,Z 736.065,A -85,B 0,C 180,E1 -10654.334,E2 -10654.334} C_VEL
LIN {X 0,Y 411.194,Z 736.073,A -85,B 0,C 180,E1 -10657.974,E2 -10657.974} C_VEL
LIN {X 0,Y 411.18,Z 736.063,A -85,B 0,C 180,E1 -10660.505,E2 -10660.505} C_VEL
LIN {X 0,Y 411.172,Z 736.044,A -85,B 0,C 180,E1 -10663.134,E2 -10663.134} C_VEL
LIN {X 0,Y 411.169,Z 736.078,A -85,B 0,C 180,E1 -10665.881,E2 -10665.881} C_VEL
LIN {X 0,Y 411.164,Z 736.078,A -85,B 0,C 180,E1 -10668.772,E2 -10668.772} C_VEL
LIN {X 0,Y 411.193,Z 736.062,A -85,B 0,C 180,E1 -10672.026,E2 -10672.026} C_VEL
LIN {X 0,Y 411.206,Z 736.08,A -85,B 0,C 180,E1 -10675.666,E2 -10675.666} C_VEL
LIN {X 0,Y 411.19,Z 736.068,A -85,B 0,C 180,E1 -10679.152,E2 -10679.152} C_VEL
LIN {X 0,Y 411.19,Z 736.076,A -85,B 0,C 180,E1 -10682.517,E2 -10682.517} C_VEL
LIN {X 0,Y 411.213,Z 736.075,A -85,B 0,C 180,E1 -10685.784,E2 -10685.784} C_VEL
LIN {X 0,Y 411.302,Z 736.215,A -85,B 0,C 180,E1 -10689.496,E2 -10689.496} C_VEL
LIN {X 0,Y 412.029,Z 741.406,A -85,B 0,C 180,E1 -10691.09,E2 -10691.09} C_VEL
LIN {X 0,Y 411.713,Z 750.251,A -85,B 0,C 180,E1 -10693.641,E2 -10693.641} C_VEL
LIN {X 0,Y 411.53,Z 754.534,A -85,B 0,C 180,E1 -10694.787,E2 -10694.787} C_VEL
LIN {X 0,Y 412.304,Z 759.13,A -85,B 0,C 180,E1 -10694.948,E2 -10694.948} C_VEL
LIN {X 0,Y 414.519,Z 772.524,A -85,B 0,C 180,E1 -10695.267,E2 -10695.267} C_VEL
LIN {X 0,Y 414.022,Z 829.981,A -85,B 0,C 180,E1 -10696.283,E2 -10696.283} C_VEL
LIN {X 0,Y 413.839,Z 839.845,A -85,B 0,C 180,E1 -10696.59,E2 -10696.59} C_VEL
LIN {X 0,Y 413.391,Z 850.976,A -85,B 0,C 180,E1 -10697.107,E2 -10697.107} C_VEL
LIN {X 0,Y 412.968,Z 861.815,A -85,B 0,C 180,E1 -10697.842,E2 -10697.842} C_VEL
LIN {X 0,Y 412.422,Z 870.212,A -85,B 0,C 180,E1 -10698.574,E2 -10698.574} C_VEL
LIN {X 0,Y 411.973,Z 878.134,A -85,B 0,C 180,E1 -10699.433,E2 -10699.433} C_VEL
LIN {X 0,Y 411.603,Z 883.823,A -85,B 0,C 180,E1 -10700.169,E2 -10700.169} C_VEL
LIN {X 0,Y 411.178,Z 890.172,A -85,B 0,C 180,E1 -10701.151,E2 -10701.151} C_VEL
LIN {X 0,Y 410.799,Z 896.616,A -85,B 0,C 180,E1 -10702.381,E2 -10702.381} C_VEL
LIN {X 0,Y 410.592,Z 901.752,A -85,B 0,C 180,E1 -10703.612,E2 -10703.612} C_VEL
LIN {X 0,Y 410.211,Z 906.513,A -85,B 0,C 180,E1 -10705.086,E2 -10705.086} C_VEL
LIN {X 0,Y 410.129,Z 908.83,A -85,B 0,C 180,E1 -10706.07,E2 -10706.07} C_VEL
LIN {X 0,Y 410.092,Z 910.594,A -85,B 0,C 180,E1 -10707.053,E2 -10707.053} C_VEL
LIN {X 0,Y 409.983,Z 912.071,A -85,B 0,C 180,E1 -10708.284,E2 -10708.284} C_VEL
LIN {X 0,Y 409.257,Z 912.732,A -85,B 0,C 180,E1 -10709.1,E2 -10709.1} C_VEL
LIN {X 0,Y 407.659,Z 913.027,A -85,B 0,C 180,E1 -10709.903,E2 -10709.903} C_VEL
LIN {X 0,Y 404.011,Z 912.601,A -85,B 0,C 180,E1 -10711.508,E2 -10711.508} C_VEL
LIN {X 0,Y 402.964,Z 911.64,A -85,B 0,C 180,E1 -10712.541,E2 -10712.541} C_VEL
LIN {X 0,Y 402.963,Z 911.426,A -85,B 0,C 180,E1 -10712.611,E2 -10712.611} C_VEL
LIN {X 0,Y 403.04,Z 909.257,A -85,B 0,C 180,E1 -10714,E2 -10714} C_VEL
LIN {X 0,Y 403.266,Z 905.522,A -85,B 0,C 180,E1 -10715.5,E2 -10715.5} C_VEL
LIN {X 0,Y 403.531,Z 901.957,A -85,B 0,C 180,E1 -10716.597,E2 -10716.597} C_VEL
LIN {X 0,Y 403.705,Z 897.271,A -85,B 0,C 180,E1 -10717.754,E2 -10717.754} C_VEL
LIN {X 0,Y 404.029,Z 892.33,A -85,B 0,C 180,E1 -10718.755,E2 -10718.755} C_VEL
LIN {X 0,Y 404.494,Z 886.364,A -85,B 0,C 180,E1 -10719.753,E2 -10719.753} C_VEL
LIN {X 0,Y 404.99,Z 879.102,A -85,B 0,C 180,E1 -10720.752,E2 -10720.752} C_VEL
LIN {X 0,Y 405.448,Z 871.34,A -85,B 0,C 180,E1 -10721.625,E2 -10721.625} C_VEL
LIN {X 0,Y 405.857,Z 864.646,A -85,B 0,C 180,E1 -10722.247,E2 -10722.247} C_VEL
LIN {X 0,Y 406.269,Z 856.466,A -85,B 0,C 180,E1 -10722.869,E2 -10722.869} C_VEL
LIN {X 0,Y 406.683,Z 848.175,A -85,B 0,C 180,E1 -10723.364,E2 -10723.364} C_VEL
LIN {X 0,Y 406.992,Z 839.218,A -85,B 0,C 180,E1 -10723.767,E2 -10723.767} C_VEL
LIN {X 0,Y 407.17,Z 830.169,A -85,B 0,C 180,E1 -10724.048,E2 -10724.048} C_VEL
LIN {X 0,Y 407.631,Z 772.18,A -85,B 0,C 180,E1 -10725.093,E2 -10725.093} C_VEL
LIN {X 0,Y 404.517,Z 754.575,A -85,B 0,C 180,E1 -10725.557,E2 -10725.557} C_VEL
LIN {X 0,Y 404.98,Z 745.433,A -85,B 0,C 180,E1 -10728.202,E2 -10728.202} C_VEL
LIN {X 0,Y 404.814,Z 740.281,A -85,B 0,C 180,E1 -10729.751,E2 -10729.751} C_VEL
LIN {X 0,Y 404.243,Z 737.032,A -85,B 0,C 180,E1 -10730.813,E2 -10730.813} C_VEL
LIN {X 0,Y 404.162,Z 736.955,A -85,B 0,C 180,E1 -10734.667,E2 -10734.667} C_VEL
LIN {X 0,Y 404.131,Z 736.956,A -85,B 0,C 180,E1 -10738.005,E2 -10738.005} C_VEL
LIN {X 0,Y 404.145,Z 736.953,A -85,B 0,C 180,E1 -10740.285,E2 -10740.285} C_VEL
LIN {X 0,Y 404.146,Z 736.953,A -85,B 0,C 180,E1 -10743.812,E2 -10743.812} C_VEL
LIN {X 0,Y 404.136,Z 736.947,A -85,B 0,C 180,E1 -10746.875,E2 -10746.875} C_VEL
LIN {X 0,Y 404.149,Z 736.942,A -85,B 0,C 180,E1 -10750.08,E2 -10750.08} C_VEL
LIN {X 0,Y 404.154,Z 736.952,A -85,B 0,C 180,E1 -10753.084,E2 -10753.084} C_VEL
LIN {X 0,Y 404.148,Z 736.939,A -85,B 0,C 180,E1 -10755.926,E2 -10755.926} C_VEL
LIN {X 0,Y 404.116,Z 736.927,A -85,B 0,C 180,E1 -10758.634,E2 -10758.634} C_VEL
LIN {X 0,Y 404.153,Z 736.949,A -85,B 0,C 180,E1 -10761.492,E2 -10761.492} C_VEL
LIN {X 0,Y 404.185,Z 736.946,A -85,B 0,C 180,E1 -10764.984,E2 -10764.984} C_VEL
LIN {X 0,Y 404.143,Z 736.95,A -85,B 0,C 180,E1 -10768.554,E2 -10768.554} C_VEL
LIN {X 0,Y 404.197,Z 736.943,A -85,B 0,C 180,E1 -10772,E2 -10772} C_VEL
LIN {X 0,Y 404.176,Z 736.944,A -85,B 0,C 180,E1 -10775.334,E2 -10775.334} C_VEL
LIN {X 0,Y 404.14,Z 736.954,A -85,B 0,C 180,E1 -10778.581,E2 -10778.581} C_VEL
LIN {X 0,Y 404.206,Z 736.932,A -85,B 0,C 180,E1 -10781.762,E2 -10781.762} C_VEL
LIN {X 0,Y 404.208,Z 736.938,A -85,B 0,C 180,E1 -10784.882,E2 -10784.882} C_VEL
LIN {X 0,Y 404.258,Z 736.938,A -85,B 0,C 180,E1 -10787.958,E2 -10787.958} C_VEL
LIN {X 0,Y 404.435,Z 736.896,A -85,B 0,C 180,E1 -10792.1,E2 -10792.1} C_VEL
LIN {X 0,Y 404.423,Z 736.91,A -85,B 0,C 180,E1 -10794.015,E2 -10794.015} C_VEL
LIN {X 0,Y 404.485,Z 736.91,A -85,B 0,C 180,E1 -10798.008,E2 -10798.008} C_VEL
LIN {X 0,Y 404.611,Z 736.887,A -85,B 0,C 180,E1 -10800,E2 -10800} C_VEL
LIN {X 0,Y 404.418,Z 736.9,A -85,B 0,C 180,E1 -10802.988,E2 -10802.988} C_VEL
LIN {X 0,Y 404.422,Z 736.92,A -85,B 0,C 180,E1 -10805.985,E2 -10805.985} C_VEL
LIN {X 0,Y 404.293,Z 736.932,A -85,B 0,C 180,E1 -10809.001,E2 -10809.001} C_VEL
LIN {X 0,Y 404.258,Z 736.924,A -85,B 0,C 180,E1 -10812.041,E2 -10812.041} C_VEL
LIN {X 0,Y 404.208,Z 736.94,A -85,B 0,C 180,E1 -10815.118,E2 -10815.118} C_VEL
LIN {X 0,Y 404.215,Z 736.943,A -85,B 0,C 180,E1 -10818.238,E2 -10818.238} C_VEL
LIN {X 0,Y 404.143,Z 736.939,A -85,B 0,C 180,E1 -10821.419,E2 -10821.419} C_VEL
LIN {X 0,Y 404.179,Z 736.948,A -85,B 0,C 180,E1 -10824.665,E2 -10824.665} C_VEL
LIN {X 0,Y 404.196,Z 736.943,A -85,B 0,C 180,E1 -10827.999,E2 -10827.999} C_VEL
LIN {X 0,Y 404.14,Z 736.95,A -85,B 0,C 180,E1 -10831.558,E2 -10831.558} C_VEL
LIN {X 0,Y 404.187,Z 736.943,A -85,B 0,C 180,E1 -10835.016,E2 -10835.016} C_VEL
LIN {X 0,Y 404.163,Z 736.912,A -85,B 0,C 180,E1 -10838.756,E2 -10838.756} C_VEL
LIN {X 0,Y 404.15,Z 736.936,A -85,B 0,C 180,E1 -10841.604,E2 -10841.604} C_VEL
LIN {X 0,Y 404.146,Z 736.958,A -85,B 0,C 180,E1 -10844.522,E2 -10844.522} C_VEL
LIN {X 0,Y 404.138,Z 736.944,A -85,B 0,C 180,E1 -10847.296,E2 -10847.296} C_VEL
LIN {X 0,Y 404.169,Z 736.942,A -85,B 0,C 180,E1 -10849.955,E2 -10849.955} C_VEL
LIN {X 0,Y 404.141,Z 736.949,A -85,B 0,C 180,E1 -10853.124,E2 -10853.124} C_VEL
LIN {X 0,Y 404.145,Z 736.955,A -85,B 0,C 180,E1 -10856.188,E2 -10856.188} C_VEL
LIN {X 0,Y 404.146,Z 736.936,A -85,B 0,C 180,E1 -10859.715,E2 -10859.715} C_VEL
LIN {X 0,Y 404.198,Z 736.938,A -85,B 0,C 180,E1 -10863.123,E2 -10863.123} C_VEL
LIN {X 0,Y 404.235,Z 737.092,A -85,B 0,C 180,E1 -10864.698,E2 -10864.698} C_VEL
LIN {X 0,Y 405.951,Z 746.408,A -85,B 0,C 180,E1 -10867.16,E2 -10867.16} C_VEL
LIN {X 0,Y 406.018,Z 750.4,A -85,B 0,C 180,E1 -10868.151,E2 -10868.151} C_VEL
LIN {X 0,Y 405.05,Z 765.467,A -85,B 0,C 180,E1 -10871.801,E2 -10871.801} C_VEL
LIN {X 0,Y 404.415,Z 776.635,A -85,B 0,C 180,E1 -10874.438,E2 -10874.438} C_VEL
LIN {X 0,Y 404.804,Z 779.701,A -85,B 0,C 180,E1 -10874.564,E2 -10874.564} C_VEL
LIN {X 0,Y 407.442,Z 798.723,A -85,B 0,C 180,E1 -10875.005,E2 -10875.005} C_VEL
LIN {X 0,Y 407.023,Z 854.186,A -85,B 0,C 180,E1 -10876.011,E2 -10876.011} C_VEL
LIN {X 0,Y 406.64,Z 864.625,A -85,B 0,C 180,E1 -10876.348,E2 -10876.348} C_VEL
LIN {X 0,Y 406.2,Z 875.318,A -85,B 0,C 180,E1 -10876.874,E2 -10876.874} C_VEL
LIN {X 0,Y 405.629,Z 885.941,A -85,B 0,C 180,E1 -10877.619,E2 -10877.619} C_VEL
LIN {X 0,Y 405.124,Z 894.264,A -85,B 0,C 180,E1 -10878.365,E2 -10878.365} C_VEL
LIN {X 0,Y 404.614,Z 902.142,A -85,B 0,C 180,E1 -10879.238,E2 -10879.238} C_VEL
LIN {X 0,Y 404.121,Z 909.509,A -85,B 0,C 180,E1 -10880.238,E2 -10880.238} C_VEL
LIN {X 0,Y 403.642,Z 916.985,A -85,B 0,C 180,E1 -10881.489,E2 -10881.489} C_VEL
LIN {X 0,Y 403.28,Z 923.814,A -85,B 0,C 180,E1 -10882.993,E2 -10882.993} C_VEL
LIN {X 0,Y 403.031,Z 929.001,A -85,B 0,C 180,E1 -10884.496,E2 -10884.496} C_VEL
LIN {X 0,Y 402.969,Z 931.653,A -85,B 0,C 180,E1 -10885.499,E2 -10885.499} C_VEL
LIN {X 0,Y 402.838,Z 934.562,A -85,B 0,C 180,E1 -10887,E2 -10887} C_VEL
LIN {X 0,Y 402.863,Z 935.818,A -85,B 0,C 180,E1 -10888.001,E2 -10888.001} C_VEL
LIN {X 0,Y 402.86,Z 936.6,A -85,B 0,C 180,E1 -10889,E2 -10889} C_VEL
LIN {X 0,Y 402.848,Z 936.895,A -85,B 0,C 180,E1 -10890,E2 -10890} C_VEL
LIN {X 0,Y 402.86,Z 936.599,A -85,B 0,C 180,E1 -10891,E2 -10891} C_VEL
LIN {X 0,Y 402.863,Z 935.814,A -85,B 0,C 180,E1 -10891.999,E2 -10891.999} C_VEL
LIN {X 0,Y 402.838,Z 934.554,A -85,B 0,C 180,E1 -10893,E2 -10893} C_VEL
LIN {X 0,Y 402.969,Z 931.643,A -85,B 0,C 180,E1 -10894.501,E2 -10894.501} C_VEL
LIN {X 0,Y 403.031,Z 928.988,A -85,B 0,C 180,E1 -10895.504,E2 -10895.504} C_VEL
LIN {X 0,Y 403.28,Z 923.796,A -85,B 0,C 180,E1 -10897.007,E2 -10897.007} C_VEL
LIN {X 0,Y 403.641,Z 916.956,A -85,B 0,C 180,E1 -10898.511,E2 -10898.511} C_VEL
LIN {X 0,Y 404.12,Z 909.482,A -85,B 0,C 180,E1 -10899.762,E2 -10899.762} C_VEL
LIN {X 0,Y 404.614,Z 902.113,A -85,B 0,C 180,E1 -10900.762,E2 -10900.762} C_VEL
LIN {X 0,Y 405.123,Z 894.223,A -85,B 0,C 180,E1 -10901.635,E2 -10901.635} C_VEL
LIN {X 0,Y 405.618,Z 885.887,A -85,B 0,C 180,E1 -10902.381,E2 -10902.381} C_VEL
LIN {X 0,Y 406.254,Z 875.248,A -85,B 0,C 180,E1 -10903.124,E2 -10903.124} C_VEL
LIN {X 0,Y 406.618,Z 863.671,A -85,B 0,C 180,E1 -10903.685,E2 -10903.685} C_VEL
LIN {X 0,Y 407.02,Z 853.993,A -85,B 0,C 180,E1 -10903.989,E2 -10903.989} C_VEL
LIN {X 0,Y 407.426,Z 798.941,A -85,B 0,C 180,E1 -10904.987,E2 -10904.987} C_VEL
LIN {X 0,Y 404.461,Z 777.092,A -85,B 0,C 180,E1 -10905.512,E2 -10905.512} C_VEL
LIN {X 0,Y 404.469,Z 775.107,A -85,B 0,C 180,E1 -10905.883,E2 -10905.883} C_VEL
LIN {X 0,Y 405.253,Z 761.167,A -85,B 0,C 180,E1 -10909.239,E2 -10909.239} C_VEL
LIN {X 0,Y 406.136,Z 748.21,A -85,B 0,C 180,E1 -10912.377,E2 -10912.377} C_VEL
LIN {X 0,Y 404.299,Z 737.384,A -85,B 0,C 180,E1 -10915.192,E2 -10915.192} C_VEL
LIN {X 0,Y 404.219,Z 736.944,A -85,B 0,C 180,E1 -10915.48,E2 -10915.48} C_VEL
LIN {X 0,Y 404.196,Z 736.95,A -85,B 0,C 180,E1 -10918,E2 -10918} C_VEL
LIN {X 0,Y 404.14,Z 736.942,A -85,B 0,C 180,E1 -10921.558,E2 -10921.558} C_VEL
LIN {X 0,Y 404.186,Z 736.948,A -85,B 0,C 180,E1 -10925.016,E2 -10925.016} C_VEL
LIN {X 0,Y 404.161,Z 736.951,A -85,B 0,C 180,E1 -10928.756,E2 -10928.756} C_VEL
LIN {X 0,Y 404.124,Z 736.944,A -85,B 0,C 180,E1 -10931.6,E2 -10931.6} C_VEL
LIN {X 0,Y 404.148,Z 736.952,A -85,B 0,C 180,E1 -10934.522,E2 -10934.522} C_VEL
LIN {X 0,Y 404.171,Z 736.946,A -85,B 0,C 180,E1 -10937.3,E2 -10937.3} C_VEL
LIN {X 0,Y 404.169,Z 736.911,A -85,B 0,C 180,E1 -10939.956,E2 -10939.956} C_VEL
LIN {X 0,Y 404.141,Z 736.937,A -85,B 0,C 180,E1 -10943.124,E2 -10943.124} C_VEL
LIN {X 0,Y 404.146,Z 736.955,A -85,B 0,C 180,E1 -10946.188,E2 -10946.188} C_VEL
LIN {X 0,Y 404.146,Z 736.947,A -85,B 0,C 180,E1 -10949.715,E2 -10949.715} C_VEL
LIN {X 0,Y 404.196,Z 736.944,A -85,B 0,C 180,E1 -10953.123,E2 -10953.123} C_VEL
LIN {X 0,Y 404.179,Z 736.948,A -85,B 0,C 180,E1 -10955.335,E2 -10955.335} C_VEL
LIN {X 0,Y 404.143,Z 736.94,A -85,B 0,C 180,E1 -10958.581,E2 -10958.581} C_VEL
LIN {X 0,Y 404.215,Z 736.943,A -85,B 0,C 180,E1 -10961.762,E2 -10961.762} C_VEL
LIN {X 0,Y 404.208,Z 736.94,A -85,B 0,C 180,E1 -10964.882,E2 -10964.882} C_VEL
LIN {X 0,Y 404.258,Z 736.923,A -85,B 0,C 180,E1 -10967.959,E2 -10967.959} C_VEL
LIN {X 0,Y 404.406,Z 736.923,A -85,B 0,C 180,E1 -10972.129,E2 -10972.129} C_VEL
LIN {X 0,Y 404.422,Z 736.92,A -85,B 0,C 180,E1 -10974.015,E2 -10974.015} C_VEL
LIN {X 0,Y 404.482,Z 736.892,A -85,B 0,C 180,E1 -10978.009,E2 -10978.009} C_VEL
LIN {X 0,Y 404.614,Z 736.887,A -85,B 0,C 180,E1 -10980,E2 -10980} C_VEL
LIN {X 0,Y 404.425,Z 736.918,A -85,B 0,C 180,E1 -10982.988,E2 -10982.988} C_VEL
LIN {X 0,Y 404.412,Z 736.902,A -85,B 0,C 180,E1 -10986.987,E2 -10986.987} C_VEL
LIN {X 0,Y 404.26,Z 736.931,A -85,B 0,C 180,E1 -10990.012,E2 -10990.012} C_VEL
LIN {X 0,Y 404.268,Z 736.938,A -85,B 0,C 180,E1 -10993.211,E2 -10993.211} C_VEL
LIN {X 0,Y 404.217,Z 736.931,A -85,B 0,C 180,E1 -10997.007,E2 -10997.007} C_VEL
LIN {X 0,Y 404.165,Z 736.948,A -85,B 0,C 180,E1 -11000.352,E2 -11000.352} C_VEL
LIN {X 0,Y 404.165,Z 736.946,A -85,B 0,C 180,E1 -11003.575,E2 -11003.575} C_VEL
LIN {X 0,Y 404.185,Z 736.933,A -85,B 0,C 180,E1 -11005.766,E2 -11005.766} C_VEL
LIN {X 0,Y 404.197,Z 736.942,A -85,B 0,C 180,E1 -11008,E2 -11008} C_VEL
LIN {X 0,Y 404.14,Z 736.95,A -85,B 0,C 180,E1 -11011.558,E2 -11011.558} C_VEL
LIN {X 0,Y 404.185,Z 736.945,A -85,B 0,C 180,E1 -11015.016,E2 -11015.016} C_VEL
LIN {X 0,Y 404.154,Z 736.95,A -85,B 0,C 180,E1 -11018.757,E2 -11018.757} C_VEL
LIN {X 0,Y 404.12,Z 736.924,A -85,B 0,C 180,E1 -11021.599,E2 -11021.599} C_VEL
LIN {X 0,Y 404.146,Z 736.938,A -85,B 0,C 180,E1 -11024.522,E2 -11024.522} C_VEL
LIN {X 0,Y 404.137,Z 736.957,A -85,B 0,C 180,E1 -11027.296,E2 -11027.296} C_VEL
LIN {X 0,Y 404.17,Z 736.941,A -85,B 0,C 180,E1 -11029.955,E2 -11029.955} C_VEL
LIN {X 0,Y 404.137,Z 736.946,A -85,B 0,C 180,E1 -11033.125,E2 -11033.125} C_VEL
LIN {X 0,Y 404.146,Z 736.953,A -85,B 0,C 180,E1 -11036.188,E2 -11036.188} C_VEL
LIN {X 0,Y 404.145,Z 736.951,A -85,B 0,C 180,E1 -11039.715,E2 -11039.715} C_VEL
LIN {X 0,Y 404.136,Z 736.955,A -85,B 0,C 180,E1 -11043.119,E2 -11043.119} C_VEL
LIN {X 0,Y 404.161,Z 736.947,A -85,B 0,C 180,E1 -11046.425,E2 -11046.425} C_VEL
LIN {X 0,Y 404.244,Z 737.058,A -85,B 0,C 180,E1 -11049.32,E2 -11049.32} C_VEL
LIN {X 0,Y 404.941,Z 741.596,A -85,B 0,C 180,E1 -11050.746,E2 -11050.746} C_VEL
LIN {X 0,Y 404.829,Z 748.662,A -85,B 0,C 180,E1 -11052.835,E2 -11052.835} C_VEL
LIN {X 0,Y 404.529,Z 754.787,A -85,B 0,C 180,E1 -11054.524,E2 -11054.524} C_VEL
LIN {X 0,Y 405.578,Z 760.69,A -85,B 0,C 180,E1 -11054.716,E2 -11054.716} C_VEL
LIN {X 0,Y 407.653,Z 772.76,A -85,B 0,C 180,E1 -11055.013,E2 -11055.013} C_VEL
LIN {X 0,Y 407.156,Z 830.208,A -85,B 0,C 180,E1 -11056.047,E2 -11056.047} C_VEL
LIN {X 0,Y 406.977,Z 839.235,A -85,B 0,C 180,E1 -11056.328,E2 -11056.328} C_VEL
LIN {X 0,Y 406.59,Z 848.793,A -85,B 0,C 180,E1 -11056.76,E2 -11056.76} C_VEL
LIN {X 0,Y 406.18,Z 858.809,A -85,B 0,C 180,E1 -11057.382,E2 -11057.382} C_VEL
LIN {X 0,Y 405.562,Z 869.198,A -85,B 0,C 180,E1 -11058.251,E2 -11058.251} C_VEL
LIN {X 0,Y 405.097,Z 877.328,A -85,B 0,C 180,E1 -11059.125,E2 -11059.125} C_VEL
LIN {X 0,Y 404.612,Z 884.035,A -85,B 0,C 180,E1 -11059.997,E2 -11059.997} C_VEL
LIN {X 0,Y 404.156,Z 890.384,A -85,B 0,C 180,E1 -11060.996,E2 -11060.996} C_VEL
LIN {X 0,Y 403.769,Z 896.826,A -85,B 0,C 180,E1 -11062.247,E2 -11062.247} C_VEL
LIN {X 0,Y 403.562,Z 901.45,A -85,B 0,C 180,E1 -11063.365,E2 -11063.365} C_VEL
LIN {X 0,Y 403.277,Z 905.237,A -85,B 0,C 180,E1 -11064.5,E2 -11064.5} C_VEL
LIN {X 0,Y 403.092,Z 907.896,A -85,B 0,C 180,E1 -11065.5,E2 -11065.5} C_VEL
LIN {X 0,Y 402.998,Z 910.804,A -85,B 0,C 180,E1 -11067.001,E2 -11067.001} C_VEL
LIN {X 0,Y 402.914,Z 912.288,A -85,B 0,C 180,E1 -11068.264,E2 -11068.264} C_VEL
LIN {X 0,Y 402.865,Z 912.881,A -85,B 0,C 180,E1 -11069,E2 -11069} C_VEL
LIN {X 0,Y 402.85,Z 913.187,A -85,B 0,C 180,E1 -11070,E2 -11070} C_VEL
LIN {X 0,Y 402.865,Z 912.911,A -85,B 0,C 180,E1 -11071,E2 -11071} C_VEL
LIN {X 0,Y 402.963,Z 911.426,A -85,B 0,C 180,E1 -11072.611,E2 -11072.611} C_VEL
LIN {X 0,Y 402.381,Z 910.309,A -85,B 0,C 180,E1 -11073.432,E2 -11073.432} C_VEL
LIN {X 0,Y 399.729,Z 907.82,A -85,B 0,C 180,E1 -11074.75,E2 -11074.75} C_VEL
LIN {X 0,Y 397.483,Z 905.185,A -85,B 0,C 180,E1 -11075.783,E2 -11075.783} C_VEL
LIN {X 0,Y 396.539,Z 902.761,A -85,B 0,C 180,E1 -11076.552,E2 -11076.552} C_VEL
LIN {X 0,Y 396.475,Z 901.825,A -85,B 0,C 180,E1 -11076.806,E2 -11076.806} C_VEL
LIN {X 0,Y 396.663,Z 897.478,A -85,B 0,C 180,E1 -11077.892,E2 -11077.892} C_VEL
LIN {X 0,Y 397.004,Z 892.537,A -85,B 0,C 180,E1 -11078.911,E2 -11078.911} C_VEL
LIN {X 0,Y 397.515,Z 886.569,A -85,B 0,C 180,E1 -11079.926,E2 -11079.926} C_VEL
LIN {X 0,Y 398.036,Z 879.306,A -85,B 0,C 180,E1 -11080.942,E2 -11080.942} C_VEL
LIN {X 0,Y 398.426,Z 872.77,A -85,B 0,C 180,E1 -11081.704,E2 -11081.704} C_VEL
LIN {X 0,Y 398.945,Z 864.848,A -85,B 0,C 180,E1 -11082.463,E2 -11082.463} C_VEL
LIN {X 0,Y 399.373,Z 856.667,A -85,B 0,C 180,E1 -11083.095,E2 -11083.095} C_VEL
LIN {X 0,Y 399.794,Z 848.374,A -85,B 0,C 180,E1 -11083.599,E2 -11083.599} C_VEL
LIN {X 0,Y 400.107,Z 839.414,A -85,B 0,C 180,E1 -11084.009,E2 -11084.009} C_VEL
LIN {X 0,Y 400.297,Z 830.447,A -85,B 0,C 180,E1 -11084.292,E2 -11084.292} C_VEL
LIN {X 0,Y 400.712,Z 772.392,A -85,B 0,C 180,E1 -11085.36,E2 -11085.36} C_VEL
LIN {X 0,Y 397.537,Z 754.771,A -85,B 0,C 180,E1 -11085.838,E2 -11085.838} C_VEL
LIN {X 0,Y 398.017,Z 745.618,A -85,B 0,C 180,E1 -11088.532,E2 -11088.532} C_VEL
LIN {X 0,Y 397.71,Z 740.798,A -85,B 0,C 180,E1 -11090.016,E2 -11090.016} C_VEL
LIN {X 0,Y 397.204,Z 737.901,A -85,B 0,C 180,E1 -11090.996,E2 -11090.996} C_VEL
LIN {X 0,Y 397.121,Z 737.827,A -85,B 0,C 180,E1 -11094.019,E2 -11094.019} C_VEL
LIN {X 0,Y 397.094,Z 737.833,A -85,B 0,C 180,E1 -11097.757,E2 -11097.757} C_VEL
LIN {X 0,Y 397.079,Z 737.826,A -85,B 0,C 180,E1 -11100.883,E2 -11100.883} C_VEL
LIN {X 0,Y 397.126,Z 737.835,A -85,B 0,C 180,E1 -11104.493,E2 -11104.493} C_VEL
LIN {X 0,Y 397.1,Z 737.815,A -85,B 0,C 180,E1 -11108.275,E2 -11108.275} C_VEL
LIN {X 0,Y 397.09,Z 737.833,A -85,B 0,C 180,E1 -11110.909,E2 -11110.909} C_VEL
LIN {X 0,Y 397.102,Z 737.829,A -85,B 0,C 180,E1 -11113.648,E2 -11113.648} C_VEL
LIN {X 0,Y 397.102,Z 737.802,A -85,B 0,C 180,E1 -11116.521,E2 -11116.521} C_VEL
LIN {X 0,Y 397.114,Z 737.817,A -85,B 0,C 180,E1 -11120.423,E2 -11120.423} C_VEL
LIN {X 0,Y 397.109,Z 737.83,A -85,B 0,C 180,E1 -11124.265,E2 -11124.265} C_VEL
LIN {X 0,Y 397.115,Z 737.821,A -85,B 0,C 180,E1 -11126.727,E2 -11126.727} C_VEL
LIN {X 0,Y 397.126,Z 737.827,A -85,B 0,C 180,E1 -11130.296,E2 -11130.296} C_VEL
LIN {X 0,Y 397.196,Z 737.818,A -85,B 0,C 180,E1 -11132.61,E2 -11132.61} C_VEL
LIN {X 0,Y 397.13,Z 737.82,A -85,B 0,C 180,E1 -11135.981,E2 -11135.981} C_VEL
LIN {X 0,Y 397.14,Z 737.823,A -85,B 0,C 180,E1 -11139.705,E2 -11139.705} C_VEL
LIN {X 0,Y 397.183,Z 737.806,A -85,B 0,C 180,E1 -11142.845,E2 -11142.845} C_VEL
LIN {X 0,Y 397.23,Z 737.813,A -85,B 0,C 180,E1 -11146.703,E2 -11146.703} C_VEL
LIN {X 0,Y 397.219,Z 737.81,A -85,B 0,C 180,E1 -11149.809,E2 -11149.809} C_VEL
LIN {X 0,Y 397.364,Z 737.778,A -85,B 0,C 180,E1 -11152.888,E2 -11152.888} C_VEL
LIN {X 0,Y 397.257,Z 737.804,A -85,B 0,C 180,E1 -11154.925,E2 -11154.925} C_VEL
LIN {X 0,Y 397.454,Z 737.786,A -85,B 0,C 180,E1 -11157.973,E2 -11157.973} C_VEL
LIN {X 0,Y 397.581,Z 737.763,A -85,B 0,C 180,E1 -11160,E2 -11160} C_VEL
LIN {X 0,Y 397.377,Z 737.776,A -85,B 0,C 180,E1 -11163.041,E2 -11163.041} C_VEL
LIN {X 0,Y 397.373,Z 737.797,A -85,B 0,C 180,E1 -11166.091,E2 -11166.091} C_VEL
LIN {X 0,Y 397.255,Z 737.81,A -85,B 0,C 180,E1 -11169.162,E2 -11169.162} C_VEL
LIN {X 0,Y 397.221,Z 737.799,A -85,B 0,C 180,E1 -11172.258,E2 -11172.258} C_VEL
LIN {X 0,Y 397.181,Z 737.818,A -85,B 0,C 180,E1 -11175.392,E2 -11175.392} C_VEL
LIN {X 0,Y 397.173,Z 737.817,A -85,B 0,C 180,E1 -11178.573,E2 -11178.573} C_VEL
LIN {X 0,Y 397.1,Z 737.818,A -85,B 0,C 180,E1 -11181.818,E2 -11181.818} C_VEL
LIN {X 0,Y 397.158,Z 737.822,A -85,B 0,C 180,E1 -11185.131,E2 -11185.131} C_VEL
LIN {X 0,Y 397.163,Z 737.823,A -85,B 0,C 180,E1 -11187.776,E2 -11187.776} C_VEL
LIN {X 0,Y 397.079,Z 737.829,A -85,B 0,C 180,E1 -11190.882,E2 -11190.882} C_VEL
LIN {X 0,Y 397.127,Z 737.826,A -85,B 0,C 180,E1 -11194.493,E2 -11194.493} C_VEL
LIN {X 0,Y 397.11,Z 737.795,A -85,B 0,C 180,E1 -11198.274,E2 -11198.274} C_VEL
LIN {X 0,Y 397.113,Z 737.806,A -85,B 0,C 180,E1 -11200.906,E2 -11200.906} C_VEL
LIN {X 0,Y 397.103,Z 737.827,A -85,B 0,C 180,E1 -11203.648,E2 -11203.648} C_VEL
LIN {X 0,Y 397.104,Z 737.827,A -85,B 0,C 180,E1 -11206.521,E2 -11206.521} C_VEL
LIN {X 0,Y 397.116,Z 737.826,A -85,B 0,C 180,E1 -11210.423,E2 -11210.423} C_VEL
LIN {X 0,Y 397.11,Z 737.823,A -85,B 0,C 180,E1 -11214.265,E2 -11214.265} C_VEL
LIN {X 0,Y 397.115,Z 737.831,A -85,B 0,C 180,E1 -11216.727,E2 -11216.727} C_VEL
LIN {X 0,Y 397.125,Z 737.816,A -85,B 0,C 180,E1 -11220.296,E2 -11220.296} C_VEL
LIN {X 0,Y 397.195,Z 737.814,A -85,B 0,C 180,E1 -11222.61,E2 -11222.61} C_VEL
LIN {X 0,Y 397.195,Z 737.934,A -85,B 0,C 180,E1 -11224.475,E2 -11224.475} C_VEL
LIN {X 0,Y 399.019,Z 748.045,A -85,B 0,C 180,E1 -11227.202,E2 -11227.202} C_VEL
LIN {X 0,Y 399.045,Z 751.296,A -85,B 0,C 180,E1 -11228.022,E2 -11228.022} C_VEL
LIN {X 0,Y 398.013,Z 766.356,A -85,B 0,C 180,E1 -11231.734,E2 -11231.734} C_VEL
LIN {X 0,Y 397.44,Z 776.433,A -85,B 0,C 180,E1 -11234.158,E2 -11234.158} C_VEL
LIN {X 0,Y 397.904,Z 779.983,A -85,B 0,C 180,E1 -11234.298,E2 -11234.298} C_VEL
LIN {X 0,Y 400.603,Z 800.204,A -85,B 0,C 180,E1 -11234.773,E2 -11234.773} C_VEL
LIN {X 0,Y 400.149,Z 853.99,A -85,B 0,C 180,E1 -11235.766,E2 -11235.766} C_VEL
LIN {X 0,Y 399.749,Z 864.425,A -85,B 0,C 180,E1 -11236.108,E2 -11236.108} C_VEL
LIN {X 0,Y 399.29,Z 875.115,A -85,B 0,C 180,E1 -11236.643,E2 -11236.643} C_VEL
LIN {X 0,Y 398.681,Z 885.735,A -85,B 0,C 180,E1 -11237.4,E2 -11237.4} C_VEL
LIN {X 0,Y 398.145,Z 894.057,A -85,B 0,C 180,E1 -11238.159,E2 -11238.159} C_VEL
LIN {X 0,Y 397.629,Z 901.935,A -85,B 0,C 180,E1 -11239.047,E2 -11239.047} C_VEL
LIN {X 0,Y 397.1,Z 909.301,A -85,B 0,C 180,E1 -11240.063,E2 -11240.063} C_VEL
LIN {X 0,Y 396.598,Z 916.777,A -85,B 0,C 180,E1 -11241.337,E2 -11241.337} C_VEL
LIN {X 0,Y 396.215,Z 923.606,A -85,B 0,C 180,E1 -11242.867,E2 -11242.867} C_VEL
LIN {X 0,Y 395.996,Z 927.266,A -85,B 0,C 180,E1 -11243.887,E2 -11243.887} C_VEL
LIN {X 0,Y 395.927,Z 930.272,A -85,B 0,C 180,E1 -11244.908,E2 -11244.908} C_VEL
LIN {X 0,Y 395.827,Z 932.602,A -85,B 0,C 180,E1 -11245.927,E2 -11245.927} C_VEL
LIN {X 0,Y 395.742,Z 934.353,A -85,B 0,C 180,E1 -11246.946,E2 -11246.946} C_VEL
LIN {X 0,Y 395.762,Z 935.61,A -85,B 0,C 180,E1 -11247.965,E2 -11247.965} C_VEL
LIN {X 0,Y 395.788,Z 936.392,A -85,B 0,C 180,E1 -11248.983,E2 -11248.983} C_VEL
LIN {X 0,Y 395.775,Z 936.687,A -85,B 0,C 180,E1 -11250,E2 -11250} C_VEL
LIN {X 0,Y 395.788,Z 936.39,A -85,B 0,C 180,E1 -11251.017,E2 -11251.017} C_VEL
LIN {X 0,Y 395.762,Z 935.605,A -85,B 0,C 180,E1 -11252.035,E2 -11252.035} C_VEL
LIN {X 0,Y 395.742,Z 934.345,A -85,B 0,C 180,E1 -11253.054,E2 -11253.054} C_VEL
LIN {X 0,Y 395.9,Z 931.434,A -85,B 0,C 180,E1 -11254.582,E2 -11254.582} C_VEL
LIN {X 0,Y 395.934,Z 928.777,A -85,B 0,C 180,E1 -11255.603,E2 -11255.603} C_VEL
LIN {X 0,Y 396.101,Z 925.509,A -85,B 0,C 180,E1 -11256.622,E2 -11256.622} C_VEL
LIN {X 0,Y 396.389,Z 920.358,A -85,B 0,C 180,E1 -11257.898,E2 -11257.898} C_VEL
LIN {X 0,Y 396.683,Z 915.327,A -85,B 0,C 180,E1 -11258.918,E2 -11258.918} C_VEL
LIN {X 0,Y 397.1,Z 909.27,A -85,B 0,C 180,E1 -11259.937,E2 -11259.937} C_VEL
LIN {X 0,Y 397.629,Z 901.901,A -85,B 0,C 180,E1 -11260.953,E2 -11260.953} C_VEL
LIN {X 0,Y 398.153,Z 894.01,A -85,B 0,C 180,E1 -11261.841,E2 -11261.841} C_VEL
LIN {X 0,Y 398.669,Z 885.674,A -85,B 0,C 180,E1 -11262.601,E2 -11262.601} C_VEL
LIN {X 0,Y 399.343,Z 875.034,A -85,B 0,C 180,E1 -11263.355,E2 -11263.355} C_VEL
LIN {X 0,Y 399.733,Z 863.454,A -85,B 0,C 180,E1 -11263.925,E2 -11263.925} C_VEL
LIN {X 0,Y 400.144,Z 853.771,A -85,B 0,C 180,E1 -11264.235,E2 -11264.235} C_VEL
LIN {X 0,Y 400.508,Z 799.122,A -85,B 0,C 180,E1 -11265.245,E2 -11265.245} C_VEL
LIN {X 0,Y 397.442,Z 776.88,A -85,B 0,C 180,E1 -11265.793,E2 -11265.793} C_VEL
LIN {X 0,Y 397.49,Z 774.902,A -85,B 0,C 180,E1 -11266.169,E2 -11266.169} C_VEL
LIN {X 0,Y 398.413,Z 759.896,A -85,B 0,C 180,E1 -11269.851,E2 -11269.851} C_VEL
LIN {X 0,Y 399.131,Z 749.108,A -85,B 0,C 180,E1 -11272.518,E2 -11272.518} C_VEL
LIN {X 0,Y 397.223,Z 738.038,A -85,B 0,C 180,E1 -11275.468,E2 -11275.468} C_VEL
LIN {X 0,Y 397.123,Z 737.832,A -85,B 0,C 180,E1 -11278.544,E2 -11278.544} C_VEL
LIN {X 0,Y 397.079,Z 737.829,A -85,B 0,C 180,E1 -11282.072,E2 -11282.072} C_VEL
LIN {X 0,Y 397.121,Z 737.824,A -85,B 0,C 180,E1 -11285.504,E2 -11285.504} C_VEL
LIN {X 0,Y 397.135,Z 737.827,A -85,B 0,C 180,E1 -11288.862,E2 -11288.862} C_VEL
LIN {X 0,Y 397.071,Z 737.826,A -85,B 0,C 180,E1 -11292.267,E2 -11292.267} C_VEL
LIN {X 0,Y 397.088,Z 737.833,A -85,B 0,C 180,E1 -11295.069,E2 -11295.069} C_VEL
LIN {X 0,Y 397.11,Z 737.814,A -85,B 0,C 180,E1 -11298.014,E2 -11298.014} C_VEL
LIN {X 0,Y 397.137,Z 737.784,A -85,B 0,C 180,E1 -11301.137,E2 -11301.137} C_VEL
LIN {X 0,Y 397.121,Z 737.824,A -85,B 0,C 180,E1 -11304.497,E2 -11304.497} C_VEL
LIN {X 0,Y 397.079,Z 737.835,A -85,B 0,C 180,E1 -11307.929,E2 -11307.929} C_VEL
LIN {X 0,Y 397.123,Z 737.817,A -85,B 0,C 180,E1 -11311.457,E2 -11311.457} C_VEL
LIN {X 0,Y 397.154,Z 737.824,A -85,B 0,C 180,E1 -11314.488,E2 -11314.488} C_VEL
LIN {X 0,Y 397.111,Z 737.821,A -85,B 0,C 180,E1 -11317.086,E2 -11317.086} C_VEL
LIN {X 0,Y 397.167,Z 737.819,A -85,B 0,C 180,E1 -11320.354,E2 -11320.354} C_VEL
LIN {X 0,Y 397.168,Z 737.822,A -85,B 0,C 180,E1 -11323.553,E2 -11323.553} C_VEL
LIN {X 0,Y 397.23,Z 737.799,A -85,B 0,C 180,E1 -11326.703,E2 -11326.703} C_VEL
LIN {X 0,Y 397.22,Z 737.807,A -85,B 0,C 180,E1 -11329.809,E2 -11329.809} C_VEL
LIN {X 0,Y 397.352,Z 737.799,A -85,B 0,C 180,E1 -11332.888,E2 -11332.888} C_VEL
LIN {X 0,Y 397.256,Z 737.805,A -85,B 0,C 180,E1 -11334.925,E2 -11334.925} C_VEL
LIN {X 0,Y 397.451,Z 737.767,A -85,B 0,C 180,E1 -11337.973,E2 -11337.973} C_VEL
LIN {X 0,Y 397.583,Z 737.762,A -85,B 0,C 180,E1 -11340,E2 -11340} C_VEL
LIN {X 0,Y 397.384,Z 737.795,A -85,B 0,C 180,E1 -11343.041,E2 -11343.041} C_VEL
LIN {X 0,Y 397.364,Z 737.778,A -85,B 0,C 180,E1 -11347.112,E2 -11347.112} C_VEL
LIN {X 0,Y 397.219,Z 737.809,A -85,B 0,C 180,E1 -11350.191,E2 -11350.191} C_VEL
LIN {X 0,Y 397.228,Z 737.814,A -85,B 0,C 180,E1 -11353.321,E2 -11353.321} C_VEL
LIN {X 0,Y 397.183,Z 737.806,A -85,B 0,C 180,E1 -11357.155,E2 -11357.155} C_VEL
LIN {X 0,Y 397.104,Z 737.831,A -85,B 0,C 180,E1 -11360.73,E2 -11360.73} C_VEL
LIN {X 0,Y 397.13,Z 737.821,A -85,B 0,C 180,E1 -11364.019,E2 -11364.019} C_VEL
LIN {X 0,Y 397.196,Z 737.816,A -85,B 0,C 180,E1 -11367.39,E2 -11367.39} C_VEL
LIN {X 0,Y 397.08,Z 737.836,A -85,B 0,C 180,E1 -11370.882,E2 -11370.882} C_VEL
LIN {X 0,Y 397.126,Z 737.819,A -85,B 0,C 180,E1 -11374.493,E2 -11374.493} C_VEL
LIN {X 0,Y 397.102,Z 737.827,A -85,B 0,C 180,E1 -11378.275,E2 -11378.275} C_VEL
LIN {X 0,Y 397.087,Z 737.812,A -85,B 0,C 180,E1 -11380.909,E2 -11380.909} C_VEL
LIN {X 0,Y 397.101,Z 737.802,A -85,B 0,C 180,E1 -11383.649,E2 -11383.649} C_VEL
LIN {X 0,Y 397.103,Z 737.828,A -85,B 0,C 180,E1 -11386.521,E2 -11386.521} C_VEL
LIN {X 0,Y 397.114,Z 737.817,A -85,B 0,C 180,E1 -11390.423,E2 -11390.423} C_VEL
LIN {X 0,Y 397.109,Z 737.832,A -85,B 0,C 180,E1 -11394.265,E2 -11394.265} C_VEL
LIN {X 0,Y 397.116,Z 737.827,A -85,B 0,C 180,E1 -11396.727,E2 -11396.727} C_VEL
LIN {X 0,Y 397.12,Z 737.83,A -85,B 0,C 180,E1 -11400.295,E2 -11400.295} C_VEL
LIN {X 0,Y 397.096,Z 737.835,A -85,B 0,C 180,E1 -11403.739,E2 -11403.739} C_VEL
LIN {X 0,Y 397.105,Z 737.827,A -85,B 0,C 180,E1 -11407.085,E2 -11407.085} C_VEL
LIN {X 0,Y 397.228,Z 738.067,A -85,B 0,C 180,E1 -11409.209,E2 -11409.209} C_VEL
LIN {X 0,Y 398.005,Z 743.535,A -85,B 0,C 180,E1 -11410.933,E2 -11410.933} C_VEL
LIN {X 0,Y 397.785,Z 750.641,A -85,B 0,C 180,E1 -11413.051,E2 -11413.051} C_VEL
LIN {X 0,Y 397.577,Z 754.951,A -85,B 0,C 180,E1 -11414.242,E2 -11414.242} C_VEL
LIN {X 0,Y 398.426,Z 759.908,A -85,B 0,C 180,E1 -11414.416,E2 -11414.416} C_VEL
LIN {X 0,Y 400.792,Z 774.082,A -85,B 0,C 180,E1 -11414.77,E2 -11414.77} C_VEL
LIN {X 0,Y 400.289,Z 830.436,A -85,B 0,C 180,E1 -11415.803,E2 -11415.803} C_VEL
LIN {X 0,Y 400.107,Z 839.456,A -85,B 0,C 180,E1 -11416.088,E2 -11416.088} C_VEL
LIN {X 0,Y 399.69,Z 849.011,A -85,B 0,C 180,E1 -11416.527,E2 -11416.527} C_VEL
LIN {X 0,Y 399.251,Z 859.025,A -85,B 0,C 180,E1 -11417.16,E2 -11417.16} C_VEL
LIN {X 0,Y 398.625,Z 869.411,A -85,B 0,C 180,E1 -11418.044,E2 -11418.044} C_VEL
LIN {X 0,Y 398.137,Z 877.54,A -85,B 0,C 180,E1 -11418.932,E2 -11418.932} C_VEL
LIN {X 0,Y 397.639,Z 884.247,A -85,B 0,C 180,E1 -11419.82,E2 -11419.82} C_VEL
LIN {X 0,Y 397.158,Z 890.595,A -85,B 0,C 180,E1 -11420.836,E2 -11420.836} C_VEL
LIN {X 0,Y 396.739,Z 897.037,A -85,B 0,C 180,E1 -11422.109,E2 -11422.109} C_VEL
LIN {X 0,Y 396.498,Z 902.05,A -85,B 0,C 180,E1 -11423.351,E2 -11423.351} C_VEL
LIN {X 0,Y 396.102,Z 906.932,A -85,B 0,C 180,E1 -11424.91,E2 -11424.91} C_VEL
LIN {X 0,Y 395.961,Z 909.25,A -85,B 0,C 180,E1 -11425.929,E2 -11425.929} C_VEL
LIN {X 0,Y 395.904,Z 911.013,A -85,B 0,C 180,E1 -11426.947,E2 -11426.947} C_VEL
LIN {X 0,Y 395.864,Z 912.285,A -85,B 0,C 180,E1 -11427.965,E2 -11427.965} C_VEL
LIN {X 0,Y 395.795,Z 913.089,A -85,B 0,C 180,E1 -11428.983,E2 -11428.983} C_VEL
LIN {X 0,Y 395.777,Z 913.395,A -85,B 0,C 180,E1 -11430,E2 -11430} C_VEL
LIN {X 0,Y 395.795,Z 913.119,A -85,B 0,C 180,E1 -11431.017,E2 -11431.017} C_VEL
LIN {X 0,Y 395.871,Z 911.674,A -85,B 0,C 180,E1 -11432.624,E2 -11432.624} C_VEL
LIN {X 0,Y 395.958,Z 909.465,A -85,B 0,C 180,E1 -11434.071,E2 -11434.071} C_VEL
LIN {X 0,Y 396.22,Z 905.729,A -85,B 0,C 180,E1 -11435.599,E2 -11435.599} C_VEL
LIN {X 0,Y 396.475,Z 901.825,A -85,B 0,C 180,E1 -11436.806,E2 -11436.806} C_VEL
LIN {X 0,Y 395.906,Z 899.099,A -85,B 0,C 180,E1 -11437.549,E2 -11437.549} C_VEL
LIN {X 0,Y 393.398,Z 894.051,A -85,B 0,C 180,E1 -11438.731,E2 -11438.731} C_VEL
LIN {X 0,Y 391.051,Z 888.283,A -85,B 0,C 180,E1 -11439.855,E2 -11439.855} C_VEL
LIN {X 0,Y 390.748,Z 884.187,A -85,B 0,C 180,E1 -11440.499,E2 -11440.499} C_VEL
LIN {X 0,Y 391.335,Z 875.392,A -85,B 0,C 180,E1 -11441.656,E2 -11441.656} C_VEL
LIN {X 0,Y 391.914,Z 866.549,A -85,B 0,C 180,E1 -11442.558,E2 -11442.558} C_VEL
LIN {X 0,Y 392.384,Z 858.738,A -85,B 0,C 180,E1 -11443.201,E2 -11443.201} C_VEL
LIN {X 0,Y 392.865,Z 849.782,A -85,B 0,C 180,E1 -11443.777,E2 -11443.777} C_VEL
LIN {X 0,Y 393.234,Z 840.44,A -85,B 0,C 180,E1 -11444.226,E2 -11444.226} C_VEL
LIN {X 0,Y 393.428,Z 830.722,A -85,B 0,C 180,E1 -11444.545,E2 -11444.545} C_VEL
LIN {X 0,Y 393.901,Z 773.44,A -85,B 0,C 180,E1 -11445.616,E2 -11445.616} C_VEL
LIN {X 0,Y 390.567,Z 755.052,A -85,B 0,C 180,E1 -11446.104,E2 -11446.104} C_VEL
LIN {X 0,Y 391.025,Z 745.804,A -85,B 0,C 180,E1 -11448.876,E2 -11448.876} C_VEL
LIN {X 0,Y 390.432,Z 740.351,A -85,B 0,C 180,E1 -11450.605,E2 -11450.605} C_VEL
LIN {X 0,Y 390.138,Z 738.774,A -85,B 0,C 180,E1 -11451.187,E2 -11451.187} C_VEL
LIN {X 0,Y 390.054,Z 738.712,A -85,B 0,C 180,E1 -11454.483,E2 -11454.483} C_VEL
LIN {X 0,Y 390.037,Z 738.712,A -85,B 0,C 180,E1 -11458.003,E2 -11458.003} C_VEL
LIN {X 0,Y 390.024,Z 738.703,A -85,B 0,C 180,E1 -11461.504,E2 -11461.504} C_VEL
LIN {X 0,Y 390.086,Z 738.707,A -85,B 0,C 180,E1 -11465.207,E2 -11465.207} C_VEL
LIN {X 0,Y 390.067,Z 738.693,A -85,B 0,C 180,E1 -11469.218,E2 -11469.218} C_VEL
LIN {X 0,Y 390.043,Z 738.713,A -85,B 0,C 180,E1 -11472.374,E2 -11472.374} C_VEL
LIN {X 0,Y 390.045,Z 738.695,A -85,B 0,C 180,E1 -11475.354,E2 -11475.354} C_VEL
LIN {X 0,Y 390.028,Z 738.674,A -85,B 0,C 180,E1 -11478.186,E2 -11478.186} C_VEL
LIN {X 0,Y 390.09,Z 738.698,A -85,B 0,C 180,E1 -11480.907,E2 -11480.907} C_VEL
LIN {X 0,Y 390.086,Z 738.704,A -85,B 0,C 180,E1 -11484.793,E2 -11484.793} C_VEL
LIN {X 0,Y 390.025,Z 738.708,A -85,B 0,C 180,E1 -11488.496,E2 -11488.496} C_VEL
LIN {X 0,Y 390.119,Z 738.696,A -85,B 0,C 180,E1 -11492.07,E2 -11492.07} C_VEL
LIN {X 0,Y 390.08,Z 738.701,A -85,B 0,C 180,E1 -11495.519,E2 -11495.519} C_VEL
LIN {X 0,Y 390.089,Z 738.703,A -85,B 0,C 180,E1 -11499.53,E2 -11499.53} C_VEL
LIN {X 0,Y 390.14,Z 738.684,A -85,B 0,C 180,E1 -11503.248,E2 -11503.248} C_VEL
LIN {X 0,Y 390.196,Z 738.689,A -85,B 0,C 180,E1 -11506.561,E2 -11506.561} C_VEL
LIN {X 0,Y 390.207,Z 738.682,A -85,B 0,C 180,E1 -11510.671,E2 -11510.671} C_VEL
LIN {X 0,Y 390.319,Z 738.654,A -85,B 0,C 180,E1 -11512.759,E2 -11512.759} C_VEL
LIN {X 0,Y 390.229,Z 738.678,A -85,B 0,C 180,E1 -11514.833,E2 -11514.833} C_VEL
LIN {X 0,Y 390.423,Z 738.662,A -85,B 0,C 180,E1 -11517.937,E2 -11517.937} C_VEL
LIN {X 0,Y 390.55,Z 738.638,A -85,B 0,C 180,E1 -11520,E2 -11520} C_VEL
LIN {X 0,Y 390.312,Z 738.656,A -85,B 0,C 180,E1 -11523.096,E2 -11523.096} C_VEL
LIN {X 0,Y 390.326,Z 738.674,A -85,B 0,C 180,E1 -11526.202,E2 -11526.202} C_VEL
LIN {X 0,Y 390.207,Z 738.69,A -85,B 0,C 180,E1 -11529.329,E2 -11529.329} C_VEL
LIN {X 0,Y 390.196,Z 738.676,A -85,B 0,C 180,E1 -11533.438,E2 -11533.438} C_VEL
LIN {X 0,Y 390.15,Z 738.696,A -85,B 0,C 180,E1 -11537.308,E2 -11537.308} C_VEL
LIN {X 0,Y 390.102,Z 738.687,A -85,B 0,C 180,E1 -11540.475,E2 -11540.475} C_VEL
LIN {X 0,Y 390.091,Z 738.697,A -85,B 0,C 180,E1 -11543.351,E2 -11543.351} C_VEL
LIN {X 0,Y 390.114,Z 738.698,A -85,B 0,C 180,E1 -11546.768,E2 -11546.768} C_VEL
LIN {X 0,Y 390.04,Z 738.703,A -85,B 0,C 180,E1 -11550.3,E2 -11550.3} C_VEL
LIN {X 0,Y 390.069,Z 738.711,A -85,B 0,C 180,E1 -11554.025,E2 -11554.025} C_VEL
LIN {X 0,Y 390.048,Z 738.688,A -85,B 0,C 180,E1 -11557.551,E2 -11557.551} C_VEL
LIN {X 0,Y 390.077,Z 738.679,A -85,B 0,C 180,E1 -11560.825,E2 -11560.825} C_VEL
LIN {X 0,Y 390.056,Z 738.706,A -85,B 0,C 180,E1 -11563.886,E2 -11563.886} C_VEL
LIN {X 0,Y 390.059,Z 738.701,A -85,B 0,C 180,E1 -11566.79,E2 -11566.79} C_VEL
LIN {X 0,Y 390.058,Z 738.698,A -85,B 0,C 180,E1 -11569.561,E2 -11569.561} C_VEL
LIN {X 0,Y 390.047,Z 738.712,A -85,B 0,C 180,E1 -11572.448,E2 -11572.448} C_VEL
LIN {X 0,Y 390.084,Z 738.706,A -85,B 0,C 180,E1 -11576.047,E2 -11576.047} C_VEL
LIN {X 0,Y 390.047,Z 738.691,A -85,B 0,C 180,E1 -11579.869,E2 -11579.869} C_VEL
LIN {X 0,Y 390.117,Z 738.691,A -85,B 0,C 180,E1 -11583.232,E2 -11583.232} C_VEL
LIN {X 0,Y 390.147,Z 738.902,A -85,B 0,C 180,E1 -11584.3,E2 -11584.3} C_VEL
LIN {X 0,Y 391.967,Z 748.937,A -85,B 0,C 180,E1 -11587.047,E2 -11587.047} C_VEL
LIN {X 0,Y 392.067,Z 752.19,A -85,B 0,C 180,E1 -11587.887,E2 -11587.887} C_VEL
LIN {X 0,Y 390.997,Z 767.226,A -85,B 0,C 180,E1 -11591.666,E2 -11591.666} C_VEL
LIN {X 0,Y 390.457,Z 776.229,A -85,B 0,C 180,E1 -11593.867,E2 -11593.867} C_VEL
LIN {X 0,Y 390.978,Z 780.324,A -85,B 0,C 180,E1 -11594.022,E2 -11594.022} C_VEL
LIN {X 0,Y 393.759,Z 801.229,A -85,B 0,C 180,E1 -11594.524,E2 -11594.524} C_VEL
LIN {X 0,Y 393.285,Z 853.796,A -85,B 0,C 180,E1 -11595.512,E2 -11595.512} C_VEL
LIN {X 0,Y 392.869,Z 864.225,A -85,B 0,C 180,E1 -11595.86,E2 -11595.86} C_VEL
LIN {X 0,Y 392.396,Z 874.912,A -85,B 0,C 180,E1 -11596.404,E2 -11596.404} C_VEL
LIN {X 0,Y 391.737,Z 885.53,A -85,B 0,C 180,E1 -11597.173,E2 -11597.173} C_VEL
LIN {X 0,Y 391.18,Z 893.851,A -85,B 0,C 180,E1 -11597.945,E2 -11597.945} C_VEL
LIN {X 0,Y 390.648,Z 901.728,A -85,B 0,C 180,E1 -11598.849,E2 -11598.849} C_VEL
LIN {X 0,Y 390.092,Z 909.094,A -85,B 0,C 180,E1 -11599.883,E2 -11599.883} C_VEL
LIN {X 0,Y 389.569,Z 916.57,A -85,B 0,C 180,E1 -11601.179,E2 -11601.179} C_VEL
LIN {X 0,Y 389.132,Z 923.397,A -85,B 0,C 180,E1 -11602.737,E2 -11602.737} C_VEL
LIN {X 0,Y 388.921,Z 927.058,A -85,B 0,C 180,E1 -11603.776,E2 -11603.776} C_VEL
LIN {X 0,Y 388.844,Z 930.064,A -85,B 0,C 180,E1 -11604.815,E2 -11604.815} C_VEL
LIN {X 0,Y 388.756,Z 932.394,A -85,B 0,C 180,E1 -11605.853,E2 -11605.853} C_VEL
LIN {X 0,Y 388.651,Z 934.145,A -85,B 0,C 180,E1 -11606.89,E2 -11606.89} C_VEL
LIN {X 0,Y 388.661,Z 935.401,A -85,B 0,C 180,E1 -11607.927,E2 -11607.927} C_VEL
LIN {X 0,Y 388.7,Z 936.184,A -85,B 0,C 180,E1 -11608.964,E2 -11608.964} C_VEL
LIN {X 0,Y 388.705,Z 936.479,A -85,B 0,C 180,E1 -11610,E2 -11610} C_VEL
LIN {X 0,Y 388.7,Z 936.182,A -85,B 0,C 180,E1 -11611.036,E2 -11611.036} C_VEL
LIN {X 0,Y 388.661,Z 935.395,A -85,B 0,C 180,E1 -11612.073,E2 -11612.073} C_VEL
LIN {X 0,Y 388.651,Z 934.135,A -85,B 0,C 180,E1 -11613.11,E2 -11613.11} C_VEL
LIN {X 0,Y 388.83,Z 931.224,A -85,B 0,C 180,E1 -11614.665,E2 -11614.665} C_VEL
LIN {X 0,Y 388.844,Z 928.567,A -85,B 0,C 180,E1 -11615.705,E2 -11615.705} C_VEL
LIN {X 0,Y 389.04,Z 925.298,A -85,B 0,C 180,E1 -11616.743,E2 -11616.743} C_VEL
LIN {X 0,Y 389.331,Z 920.147,A -85,B 0,C 180,E1 -11618.042,E2 -11618.042} C_VEL
LIN {X 0,Y 389.656,Z 915.116,A -85,B 0,C 180,E1 -11619.08,E2 -11619.08} C_VEL
LIN {X 0,Y 390.092,Z 909.058,A -85,B 0,C 180,E1 -11620.117,E2 -11620.117} C_VEL
LIN {X 0,Y 390.648,Z 901.689,A -85,B 0,C 180,E1 -11621.151,E2 -11621.151} C_VEL
LIN {X 0,Y 391.188,Z 893.798,A -85,B 0,C 180,E1 -11622.055,E2 -11622.055} C_VEL
LIN {X 0,Y 391.755,Z 885.462,A -85,B 0,C 180,E1 -11622.827,E2 -11622.827} C_VEL
LIN {X 0,Y 392.401,Z 874.818,A -85,B 0,C 180,E1 -11623.596,E2 -11623.596} C_VEL
LIN {X 0,Y 392.858,Z 863.237,A -85,B 0,C 180,E1 -11624.174,E2 -11624.174} C_VEL
LIN {X 0,Y 393.272,Z 853.549,A -85,B 0,C 180,E1 -11624.489,E2 -11624.489} C_VEL
LIN {X 0,Y 393.696,Z 800.088,A -85,B 0,C 180,E1 -11625.493,E2 -11625.493} C_VEL
LIN {X 0,Y 390.452,Z 776.575,A -85,B 0,C 180,E1 -11626.09,E2 -11626.09} C_VEL
LIN {X 0,Y 390.545,Z 773.626,A -85,B 0,C 180,E1 -11626.734,E2 -11626.734} C_VEL
LIN {X 0,Y 391.4,Z 760.783,A -85,B 0,C 180,E1 -11629.948,E2 -11629.948} C_VEL
LIN {X 0,Y 392.138,Z 750.002,A -85,B 0,C 180,E1 -11632.664,E2 -11632.664} C_VEL
LIN {X 0,Y 390.195,Z 739.135,A -85,B 0,C 180,E1 -11635.612,E2 -11635.612} C_VEL
LIN {X 0,Y 390.111,Z 738.695,A -85,B 0,C 180,E1 -11635.92,E2 -11635.92} C_VEL
LIN {X 0,Y 390.059,Z 738.704,A -85,B 0,C 180,E1 -11639.11,E2 -11639.11} C_VEL
LIN {X 0,Y 390.043,Z 738.708,A -85,B 0,C 180,E1 -11642.722,E2 -11642.722} C_VEL
LIN {X 0,Y 390.058,Z 738.702,A -85,B 0,C 180,E1 -11645.826,E2 -11645.826} C_VEL
LIN {X 0,Y 390.073,Z 738.708,A -85,B 0,C 180,E1 -11649.219,E2 -11649.219} C_VEL
LIN {X 0,Y 390.044,Z 738.7,A -85,B 0,C 180,E1 -11652.374,E2 -11652.374} C_VEL
LIN {X 0,Y 390.045,Z 738.713,A -85,B 0,C 180,E1 -11655.355,E2 -11655.355} C_VEL
LIN {X 0,Y 390.069,Z 738.689,A -85,B 0,C 180,E1 -11658.192,E2 -11658.192} C_VEL
LIN {X 0,Y 390.095,Z 738.659,A -85,B 0,C 180,E1 -11660.908,E2 -11660.908} C_VEL
LIN {X 0,Y 390.087,Z 738.699,A -85,B 0,C 180,E1 -11664.793,E2 -11664.793} C_VEL
LIN {X 0,Y 390.033,Z 738.713,A -85,B 0,C 180,E1 -11667.875,E2 -11667.875} C_VEL
LIN {X 0,Y 390.059,Z 738.695,A -85,B 0,C 180,E1 -11670.891,E2 -11670.891} C_VEL
LIN {X 0,Y 390.12,Z 738.703,A -85,B 0,C 180,E1 -11674.257,E2 -11674.257} C_VEL
LIN {X 0,Y 390.043,Z 738.7,A -85,B 0,C 180,E1 -11677.766,E2 -11677.766} C_VEL
LIN {X 0,Y 390.118,Z 738.696,A -85,B 0,C 180,E1 -11681.079,E2 -11681.079} C_VEL
LIN {X 0,Y 390.141,Z 738.697,A -85,B 0,C 180,E1 -11684.323,E2 -11684.323} C_VEL
LIN {X 0,Y 390.172,Z 738.676,A -85,B 0,C 180,E1 -11687.517,E2 -11687.517} C_VEL
LIN {X 0,Y 390.207,Z 738.69,A -85,B 0,C 180,E1 -11690.671,E2 -11690.671} C_VEL
LIN {X 0,Y 390.327,Z 738.674,A -85,B 0,C 180,E1 -11693.798,E2 -11693.798} C_VEL
LIN {X 0,Y 390.42,Z 738.642,A -85,B 0,C 180,E1 -11697.937,E2 -11697.937} C_VEL
LIN {X 0,Y 390.552,Z 738.638,A -85,B 0,C 180,E1 -11700,E2 -11700} C_VEL
LIN {X 0,Y 390.318,Z 738.675,A -85,B 0,C 180,E1 -11703.097,E2 -11703.097} C_VEL
LIN {X 0,Y 390.311,Z 738.661,A -85,B 0,C 180,E1 -11706.585,E2 -11706.585} C_VEL
LIN {X 0,Y 390.316,Z 738.656,A -85,B 0,C 180,E1 -11708.282,E2 -11708.282} C_VEL
LIN {X 0,Y 390.173,Z 738.696,A -85,B 0,C 180,E1 -11712.483,E2 -11712.483} C_VEL
LIN {X 0,Y 390.141,Z 738.687,A -85,B 0,C 180,E1 -11715.677,E2 -11715.677} C_VEL
LIN {X 0,Y 390.104,Z 738.695,A -85,B 0,C 180,E1 -11718.922,E2 -11718.922} C_VEL
LIN {X 0,Y 390.039,Z 738.709,A -85,B 0,C 180,E1 -11722.234,E2 -11722.234} C_VEL
LIN {X 0,Y 390.12,Z 738.684,A -85,B 0,C 180,E1 -11725.743,E2 -11725.743} C_VEL
LIN {X 0,Y 390.06,Z 738.711,A -85,B 0,C 180,E1 -11729.11,E2 -11729.11} C_VEL
LIN {X 0,Y 390.044,Z 738.705,A -85,B 0,C 180,E1 -11732.722,E2 -11732.722} C_VEL
LIN {X 0,Y 390.057,Z 738.708,A -85,B 0,C 180,E1 -11735.825,E2 -11735.825} C_VEL
LIN {X 0,Y 390.069,Z 738.701,A -85,B 0,C 180,E1 -11739.218,E2 -11739.218} C_VEL
LIN {X 0,Y 390.039,Z 738.669,A -85,B 0,C 180,E1 -11742.373,E2 -11742.373} C_VEL
LIN {X 0,Y 390.045,Z 738.7,A -85,B 0,C 180,E1 -11745.354,E2 -11745.354} C_VEL
LIN {X 0,Y 390.032,Z 738.711,A -85,B 0,C 180,E1 -11748.187,E2 -11748.187} C_VEL
LIN {X 0,Y 390.088,Z 738.691,A -85,B 0,C 180,E1 -11750.907,E2 -11750.907} C_VEL
LIN {X 0,Y 390.086,Z 738.706,A -85,B 0,C 180,E1 -11754.793,E2 -11754.793} C_VEL
LIN {X 0,Y 390.024,Z 738.702,A -85,B 0,C 180,E1 -11758.496,E2 -11758.496} C_VEL
LIN {X 0,Y 390.04,Z 738.711,A -85,B 0,C 180,E1 -11762.064,E2 -11762.064} C_VEL
LIN {X 0,Y 390.062,Z 738.712,A -85,B 0,C 180,E1 -11765.518,E2 -11765.518} C_VEL
LIN {X 0,Y 390.157,Z 738.874,A -85,B 0,C 180,E1 -11769.009,E2 -11769.009} C_VEL
LIN {X 0,Y 390.929,Z 743.726,A -85,B 0,C 180,E1 -11770.574,E2 -11770.574} C_VEL
LIN {X 0,Y 390.815,Z 751.071,A -85,B 0,C 180,E1 -11772.811,E2 -11772.811} C_VEL
LIN {X 0,Y 390.585,Z 755.069,A -85,B 0,C 180,E1 -11773.939,E2 -11773.939} C_VEL
LIN {X 0,Y 391.128,Z 758.27,A -85,B 0,C 180,E1 -11774.082,E2 -11774.082} C_VEL
LIN {X 0,Y 393.957,Z 774.858,A -85,B 0,C 180,E1 -11774.509,E2 -11774.509} C_VEL
LIN {X 0,Y 393.429,Z 830.664,A -85,B 0,C 180,E1 -11775.55,E2 -11775.55} C_VEL
LIN {X 0,Y 393.244,Z 839.676,A -85,B 0,C 180,E1 -11775.841,E2 -11775.841} C_VEL
LIN {X 0,Y 392.807,Z 849.228,A -85,B 0,C 180,E1 -11776.287,E2 -11776.287} C_VEL
LIN {X 0,Y 392.353,Z 859.24,A -85,B 0,C 180,E1 -11776.93,E2 -11776.93} C_VEL
LIN {X 0,Y 391.694,Z 869.625,A -85,B 0,C 180,E1 -11777.829,E2 -11777.829} C_VEL
LIN {X 0,Y 391.175,Z 877.753,A -85,B 0,C 180,E1 -11778.733,E2 -11778.733} C_VEL
LIN {X 0,Y 390.676,Z 884.458,A -85,B 0,C 180,E1 -11779.636,E2 -11779.636} C_VEL
LIN {X 0,Y 390.169,Z 890.806,A -85,B 0,C 180,E1 -11780.67,E2 -11780.67} C_VEL
LIN {X 0,Y 389.696,Z 897.249,A -85,B 0,C 180,E1 -11781.966,E2 -11781.966} C_VEL
LIN {X 0,Y 389.409,Z 902.666,A -85,B 0,C 180,E1 -11783.34,E2 -11783.34} C_VEL
LIN {X 0,Y 389.052,Z 907.142,A -85,B 0,C 180,E1 -11784.818,E2 -11784.818} C_VEL
LIN {X 0,Y 388.884,Z 909.46,A -85,B 0,C 180,E1 -11785.855,E2 -11785.855} C_VEL
LIN {X 0,Y 388.811,Z 911.223,A -85,B 0,C 180,E1 -11786.892,E2 -11786.892} C_VEL
LIN {X 0,Y 388.782,Z 912.494,A -85,B 0,C 180,E1 -11787.928,E2 -11787.928} C_VEL
LIN {X 0,Y 388.727,Z 913.297,A -85,B 0,C 180,E1 -11788.964,E2 -11788.964} C_VEL
LIN {X 0,Y 388.706,Z 913.603,A -85,B 0,C 180,E1 -11790,E2 -11790} C_VEL
LIN {X 0,Y 388.727,Z 913.327,A -85,B 0,C 180,E1 -11791.036,E2 -11791.036} C_VEL
LIN {X 0,Y 388.767,Z 912.583,A -85,B 0,C 180,E1 -11792.072,E2 -11792.072} C_VEL
LIN {X 0,Y 388.81,Z 911.373,A -85,B 0,C 180,E1 -11793.109,E2 -11793.109} C_VEL
LIN {X 0,Y 388.95,Z 908.528,A -85,B 0,C 180,E1 -11794.664,E2 -11794.664} C_VEL
LIN {X 0,Y 389.156,Z 905.936,A -85,B 0,C 180,E1 -11795.7,E2 -11795.7} C_VEL
LIN {X 0,Y 389.407,Z 901.94,A -85,B 0,C 180,E1 -11796.955,E2 -11796.955} C_VEL
LIN {X 0,Y 389.724,Z 896.517,A -85,B 0,C 180,E1 -11798.295,E2 -11798.295} C_VEL
LIN {X 0,Y 390.12,Z 891.329,A -85,B 0,C 180,E1 -11799.331,E2 -11799.331} C_VEL
LIN {X 0,Y 390.671,Z 885.076,A -85,B 0,C 180,E1 -11800.364,E2 -11800.364} C_VEL
LIN {X 0,Y 390.748,Z 884.187,A -85,B 0,C 180,E1 -11800.499,E2 -11800.499} C_VEL
LIN {X 0,Y 390.437,Z 880.031,A -85,B 0,C 180,E1 -11801.116,E2 -11801.116} C_VEL
LIN {X 0,Y 388.13,Z 872.915,A -85,B 0,C 180,E1 -11802.078,E2 -11802.078} C_VEL
LIN {X 0,Y 385.795,Z 865.179,A -85,B 0,C 180,E1 -11802.929,E2 -11802.929} C_VEL
LIN {X 0,Y 385.43,Z 860.053,A -85,B 0,C 180,E1 -11803.36,E2 -11803.36} C_VEL
LIN {X 0,Y 386.002,Z 849.981,A -85,B 0,C 180,E1 -11804.027,E2 -11804.027} C_VEL
LIN {X 0,Y 386.362,Z 840.637,A -85,B 0,C 180,E1 -11804.484,E2 -11804.484} C_VEL
LIN {X 0,Y 386.569,Z 830.994,A -85,B 0,C 180,E1 -11804.807,E2 -11804.807} C_VEL
LIN {X 0,Y 387.056,Z 774.035,A -85,B 0,C 180,E1 -11805.892,E2 -11805.892} C_VEL
LIN {X 0,Y 383.602,Z 755.177,A -85,B 0,C 180,E1 -11806.429,E2 -11806.429} C_VEL
LIN {X 0,Y 384.014,Z 747.774,A -85,B 0,C 180,E1 -11808.68,E2 -11808.68} C_VEL
LIN {X 0,Y 383.588,Z 742.456,A -85,B 0,C 180,E1 -11810.372,E2 -11810.372} C_VEL
LIN {X 0,Y 383.101,Z 739.654,A -85,B 0,C 180,E1 -11811.361,E2 -11811.361} C_VEL
LIN {X 0,Y 383.018,Z 739.588,A -85,B 0,C 180,E1 -11814.963,E2 -11814.963} C_VEL
LIN {X 0,Y 382.987,Z 739.591,A -85,B 0,C 180,E1 -11818.497,E2 -11818.497} C_VEL
LIN {X 0,Y 383.01,Z 739.576,A -85,B 0,C 180,E1 -11822.15,E2 -11822.15} C_VEL
LIN {X 0,Y 383.019,Z 739.591,A -85,B 0,C 180,E1 -11824.668,E2 -11824.668} C_VEL
LIN {X 0,Y 382.999,Z 739.572,A -85,B 0,C 180,E1 -11827.903,E2 -11827.903} C_VEL
LIN {X 0,Y 382.985,Z 739.588,A -85,B 0,C 180,E1 -11831.347,E2 -11831.347} C_VEL
LIN {X 0,Y 382.997,Z 739.586,A -85,B 0,C 180,E1 -11834.303,E2 -11834.303} C_VEL
LIN {X 0,Y 383.011,Z 739.546,A -85,B 0,C 180,E1 -11837.24,E2 -11837.24} C_VEL
LIN {X 0,Y 383.015,Z 739.573,A -85,B 0,C 180,E1 -11840.414,E2 -11840.414} C_VEL
LIN {X 0,Y 383.026,Z 739.583,A -85,B 0,C 180,E1 -11844.044,E2 -11844.044} C_VEL
LIN {X 0,Y 382.988,Z 739.582,A -85,B 0,C 180,E1 -11847.578,E2 -11847.578} C_VEL
LIN {X 0,Y 382.994,Z 739.588,A -85,B 0,C 180,E1 -11850.3,E2 -11850.3} C_VEL
LIN {X 0,Y 383.082,Z 739.561,A -85,B 0,C 180,E1 -11854.021,E2 -11854.021} C_VEL
LIN {X 0,Y 382.997,Z 739.59,A -85,B 0,C 180,E1 -11857.334,E2 -11857.334} C_VEL
LIN {X 0,Y 383.06,Z 739.578,A -85,B 0,C 180,E1 -11860.716,E2 -11860.716} C_VEL
LIN {X 0,Y 383.083,Z 739.566,A -85,B 0,C 180,E1 -11864.027,E2 -11864.027} C_VEL
LIN {X 0,Y 383.138,Z 739.575,A -85,B 0,C 180,E1 -11867.284,E2 -11867.284} C_VEL
LIN {X 0,Y 383.153,Z 739.56,A -85,B 0,C 180,E1 -11870.498,E2 -11870.498} C_VEL
LIN {X 0,Y 383.274,Z 739.53,A -85,B 0,C 180,E1 -11872.625,E2 -11872.625} C_VEL
LIN {X 0,Y 383.201,Z 739.553,A -85,B 0,C 180,E1 -11874.738,E2 -11874.738} C_VEL
LIN {X 0,Y 383.39,Z 739.538,A -85,B 0,C 180,E1 -11877.899,E2 -11877.899} C_VEL
LIN {X 0,Y 383.519,Z 739.514,A -85,B 0,C 180,E1 -11880,E2 -11880} C_VEL
LIN {X 0,Y 383.249,Z 739.536,A -85,B 0,C 180,E1 -11883.154,E2 -11883.154} C_VEL
LIN {X 0,Y 383.283,Z 739.551,A -85,B 0,C 180,E1 -11886.316,E2 -11886.316} C_VEL
LIN {X 0,Y 383.153,Z 739.568,A -85,B 0,C 180,E1 -11889.502,E2 -11889.502} C_VEL
LIN {X 0,Y 383.127,Z 739.557,A -85,B 0,C 180,E1 -11893.536,E2 -11893.536} C_VEL
LIN {X 0,Y 383.097,Z 739.576,A -85,B 0,C 180,E1 -11897.455,E2 -11897.455} C_VEL
LIN {X 0,Y 383.042,Z 739.565,A -85,B 0,C 180,E1 -11900.652,E2 -11900.652} C_VEL
LIN {X 0,Y 383.035,Z 739.58,A -85,B 0,C 180,E1 -11903.807,E2 -11903.807} C_VEL
LIN {X 0,Y 383.057,Z 739.577,A -85,B 0,C 180,E1 -11907.302,E2 -11907.302} C_VEL
LIN {X 0,Y 382.984,Z 739.585,A -85,B 0,C 180,E1 -11910.918,E2 -11910.918} C_VEL
LIN {X 0,Y 383.019,Z 739.581,A -85,B 0,C 180,E1 -11914.668,E2 -11914.668} C_VEL
LIN {X 0,Y 383.004,Z 739.556,A -85,B 0,C 180,E1 -11917.904,E2 -11917.904} C_VEL
LIN {X 0,Y 383.014,Z 739.567,A -85,B 0,C 180,E1 -11921.343,E2 -11921.343} C_VEL
LIN {X 0,Y 382.997,Z 739.59,A -85,B 0,C 180,E1 -11924.303,E2 -11924.303} C_VEL
LIN {X 0,Y 383.01,Z 739.576,A -85,B 0,C 180,E1 -11927.24,E2 -11927.24} C_VEL
LIN {X 0,Y 383.018,Z 739.581,A -85,B 0,C 180,E1 -11930.413,E2 -11930.413} C_VEL
LIN {X 0,Y 383.027,Z 739.577,A -85,B 0,C 180,E1 -11934.045,E2 -11934.045} C_VEL
LIN {X 0,Y 382.987,Z 739.584,A -85,B 0,C 180,E1 -11937.578,E2 -11937.578} C_VEL
LIN {X 0,Y 382.992,Z 739.574,A -85,B 0,C 180,E1 -11940.3,E2 -11940.3} C_VEL
LIN {X 0,Y 383.059,Z 739.573,A -85,B 0,C 180,E1 -11942.698,E2 -11942.698} C_VEL
LIN {X 0,Y 383.102,Z 739.742,A -85,B 0,C 180,E1 -11944.063,E2 -11944.063} C_VEL
LIN {X 0,Y 384.752,Z 748.74,A -85,B 0,C 180,E1 -11946.591,E2 -11946.591} C_VEL
LIN {X 0,Y 385.215,Z 752.004,A -85,B 0,C 180,E1 -11947.472,E2 -11947.472} C_VEL
LIN {X 0,Y 383.981,Z 768.1,A -85,B 0,C 180,E1 -11951.595,E2 -11951.595} C_VEL
LIN {X 0,Y 383.49,Z 776.026,A -85,B 0,C 180,E1 -11953.566,E2 -11953.566} C_VEL
LIN {X 0,Y 384.041,Z 780.184,A -85,B 0,C 180,E1 -11953.727,E2 -11953.727} C_VEL
LIN {X 0,Y 386.929,Z 802.129,A -85,B 0,C 180,E1 -11954.265,E2 -11954.265} C_VEL
LIN {X 0,Y 386.436,Z 852.555,A -85,B 0,C 180,E1 -11955.222,E2 -11955.222} C_VEL
LIN {X 0,Y 386.116,Z 861.53,A -85,B 0,C 180,E1 -11955.506,E2 -11955.506} C_VEL
LIN {X 0,Y 385.653,Z 871.198,A -85,B 0,C 180,E1 -11955.96,E2 -11955.96} C_VEL
LIN {X 0,Y 385.197,Z 880.367,A -85,B 0,C 180,E1 -11956.548,E2 -11956.548} C_VEL
LIN {X 0,Y 384.423,Z 891.179,A -85,B 0,C 180,E1 -11957.461,E2 -11957.461} C_VEL
LIN {X 0,Y 383.804,Z 899.474,A -85,B 0,C 180,E1 -11958.38,E2 -11958.38} C_VEL
LIN {X 0,Y 383.225,Z 907.178,A -85,B 0,C 180,E1 -11959.433,E2 -11959.433} C_VEL
LIN {X 0,Y 382.757,Z 913.521,A -85,B 0,C 180,E1 -11960.488,E2 -11960.488} C_VEL
LIN {X 0,Y 382.353,Z 918.792,A -85,B 0,C 180,E1 -11961.544,E2 -11961.544} C_VEL
LIN {X 0,Y 382.068,Z 923.189,A -85,B 0,C 180,E1 -11962.602,E2 -11962.602} C_VEL
LIN {X 0,Y 381.771,Z 928.075,A -85,B 0,C 180,E1 -11964.085,E2 -11964.085} C_VEL
LIN {X 0,Y 381.742,Z 931.029,A -85,B 0,C 180,E1 -11965.248,E2 -11965.248} C_VEL
LIN {X 0,Y 381.564,Z 933.936,A -85,B 0,C 180,E1 -11966.832,E2 -11966.832} C_VEL
LIN {X 0,Y 381.56,Z 935.192,A -85,B 0,C 180,E1 -11967.889,E2 -11967.889} C_VEL
LIN {X 0,Y 381.615,Z 935.975,A -85,B 0,C 180,E1 -11968.945,E2 -11968.945} C_VEL
LIN {X 0,Y 381.636,Z 936.271,A -85,B 0,C 180,E1 -11970,E2 -11970} C_VEL
LIN {X 0,Y 381.615,Z 935.973,A -85,B 0,C 180,E1 -11971.055,E2 -11971.055} C_VEL
LIN {X 0,Y 381.56,Z 935.186,A -85,B 0,C 180,E1 -11972.111,E2 -11972.111} C_VEL
LIN {X 0,Y 381.564,Z 933.926,A -85,B 0,C 180,E1 -11973.168,E2 -11973.168} C_VEL
LIN {X 0,Y 381.742,Z 931.014,A -85,B 0,C 180,E1 -11974.752,E2 -11974.752} C_VEL
LIN {X 0,Y 381.771,Z 928.057,A -85,B 0,C 180,E1 -11975.915,E2 -11975.915} C_VEL
LIN {X 0,Y 382.068,Z 923.163,A -85,B 0,C 180,E1 -11977.398,E2 -11977.398} C_VEL
LIN {X 0,Y 382.526,Z 916.322,A -85,B 0,C 180,E1 -11978.984,E2 -11978.984} C_VEL
LIN {X 0,Y 383.095,Z 908.847,A -85,B 0,C 180,E1 -11980.304,E2 -11980.304} C_VEL
LIN {X 0,Y 383.656,Z 901.476,A -85,B 0,C 180,E1 -11981.357,E2 -11981.357} C_VEL
LIN {X 0,Y 384.252,Z 893.586,A -85,B 0,C 180,E1 -11982.276,E2 -11982.276} C_VEL
LIN {X 0,Y 384.845,Z 885.249,A -85,B 0,C 180,E1 -11983.061,E2 -11983.061} C_VEL
LIN {X 0,Y 385.505,Z 874.604,A -85,B 0,C 180,E1 -11983.844,E2 -11983.844} C_VEL
LIN {X 0,Y 385.988,Z 863.019,A -85,B 0,C 180,E1 -11984.431,E2 -11984.431} C_VEL
LIN {X 0,Y 386.408,Z 853.326,A -85,B 0,C 180,E1 -11984.752,E2 -11984.752} C_VEL
LIN {X 0,Y 386.9,Z 801.062,A -85,B 0,C 180,E1 -11985.749,E2 -11985.749} C_VEL
LIN {X 0,Y 383.492,Z 776.363,A -85,B 0,C 180,E1 -11986.39,E2 -11986.39} C_VEL
LIN {X 0,Y 383.586,Z 773.422,A -85,B 0,C 180,E1 -11987.047,E2 -11987.047} C_VEL
LIN {X 0,Y 384.398,Z 761.667,A -85,B 0,C 180,E1 -11990.048,E2 -11990.048} C_VEL
LIN {X 0,Y 385.159,Z 751.979,A -85,B 0,C 180,E1 -11992.531,E2 -11992.531} C_VEL
LIN {X 0,Y 383.806,Z 743.292,A -85,B 0,C 180,E1 -11994.908,E2 -11994.908} C_VEL
LIN {X 0,Y 383.075,Z 739.614,A -85,B 0,C 180,E1 -11996.004,E2 -11996.004} C_VEL
LIN {X 0,Y 383.041,Z 739.586,A -85,B 0,C 180,E1 -11998.493,E2 -11998.493} C_VEL
LIN {X 0,Y 383.01,Z 739.581,A -85,B 0,C 180,E1 -12002.15,E2 -12002.15} C_VEL
LIN {X 0,Y 383.019,Z 739.587,A -85,B 0,C 180,E1 -12004.668,E2 -12004.668} C_VEL
LIN {X 0,Y 383.003,Z 739.589,A -85,B 0,C 180,E1 -12007.904,E2 -12007.904} C_VEL
LIN {X 0,Y 382.985,Z 739.574,A -85,B 0,C 180,E1 -12011.347,E2 -12011.347} C_VEL
LIN {X 0,Y 382.997,Z 739.587,A -85,B 0,C 180,E1 -12014.304,E2 -12014.304} C_VEL
LIN {X 0,Y 383.04,Z 739.577,A -85,B 0,C 180,E1 -12017.244,E2 -12017.244} C_VEL
LIN {X 0,Y 383.022,Z 739.538,A -85,B 0,C 180,E1 -12020.412,E2 -12020.412} C_VEL
LIN {X 0,Y 383.028,Z 739.576,A -85,B 0,C 180,E1 -12024.045,E2 -12024.045} C_VEL
LIN {X 0,Y 382.988,Z 739.592,A -85,B 0,C 180,E1 -12027.578,E2 -12027.578} C_VEL
LIN {X 0,Y 382.992,Z 739.576,A -85,B 0,C 180,E1 -12030.3,E2 -12030.3} C_VEL
LIN {X 0,Y 383.081,Z 739.582,A -85,B 0,C 180,E1 -12034.021,E2 -12034.021} C_VEL
LIN {X 0,Y 383.011,Z 739.578,A -85,B 0,C 180,E1 -12037.335,E2 -12037.335} C_VEL
LIN {X 0,Y 383.074,Z 739.574,A -85,B 0,C 180,E1 -12040.717,E2 -12040.717} C_VEL
LIN {X 0,Y 383.083,Z 739.581,A -85,B 0,C 180,E1 -12044.027,E2 -12044.027} C_VEL
LIN {X 0,Y 383.138,Z 739.551,A -85,B 0,C 180,E1 -12047.284,E2 -12047.284} C_VEL
LIN {X 0,Y 383.153,Z 739.567,A -85,B 0,C 180,E1 -12050.498,E2 -12050.498} C_VEL
LIN {X 0,Y 383.283,Z 739.551,A -85,B 0,C 180,E1 -12053.684,E2 -12053.684} C_VEL
LIN {X 0,Y 383.388,Z 739.517,A -85,B 0,C 180,E1 -12057.899,E2 -12057.899} C_VEL
LIN {X 0,Y 383.522,Z 739.513,A -85,B 0,C 180,E1 -12060,E2 -12060} C_VEL
LIN {X 0,Y 383.254,Z 739.554,A -85,B 0,C 180,E1 -12063.154,E2 -12063.154} C_VEL
LIN {X 0,Y 383.272,Z 739.538,A -85,B 0,C 180,E1 -12066.578,E2 -12066.578} C_VEL
LIN {X 0,Y 383.262,Z 739.536,A -85,B 0,C 180,E1 -12068.436,E2 -12068.436} C_VEL
LIN {X 0,Y 383.099,Z 739.573,A -85,B 0,C 180,E1 -12071.642,E2 -12071.642} C_VEL
LIN {X 0,Y 383.112,Z 739.568,A -85,B 0,C 180,E1 -12074.882,E2 -12074.882} C_VEL
LIN {X 0,Y 383.054,Z 739.565,A -85,B 0,C 180,E1 -12078.174,E2 -12078.174} C_VEL
LIN {X 0,Y 382.994,Z 739.588,A -85,B 0,C 180,E1 -12081.531,E2 -12081.531} C_VEL
LIN {X 0,Y 383.052,Z 739.57,A -85,B 0,C 180,E1 -12084.96,E2 -12084.96} C_VEL
LIN {X 0,Y 383.031,Z 739.579,A -85,B 0,C 180,E1 -12088.27,E2 -12088.27} C_VEL
LIN {X 0,Y 383.01,Z 739.579,A -85,B 0,C 180,E1 -12092.15,E2 -12092.15} C_VEL
LIN {X 0,Y 383.019,Z 739.577,A -85,B 0,C 180,E1 -12094.668,E2 -12094.668} C_VEL
LIN {X 0,Y 383,Z 739.585,A -85,B 0,C 180,E1 -12097.904,E2 -12097.904} C_VEL
LIN {X 0,Y 382.982,Z 739.558,A -85,B 0,C 180,E1 -12101.348,E2 -12101.348} C_VEL
LIN {X 0,Y 382.997,Z 739.572,A -85,B 0,C 180,E1 -12104.303,E2 -12104.303} C_VEL
LIN {X 0,Y 383.011,Z 739.588,A -85,B 0,C 180,E1 -12107.24,E2 -12107.24} C_VEL
LIN {X 0,Y 383.015,Z 739.573,A -85,B 0,C 180,E1 -12110.414,E2 -12110.414} C_VEL
LIN {X 0,Y 383.026,Z 739.588,A -85,B 0,C 180,E1 -12114.044,E2 -12114.044} C_VEL
LIN {X 0,Y 382.987,Z 739.581,A -85,B 0,C 180,E1 -12117.578,E2 -12117.578} C_VEL
LIN {X 0,Y 382.982,Z 739.591,A -85,B 0,C 180,E1 -12120.299,E2 -12120.299} C_VEL
LIN {X 0,Y 383.015,Z 739.587,A -85,B 0,C 180,E1 -12124.042,E2 -12124.042} C_VEL
LIN {X 0,Y 383.002,Z 739.586,A -85,B 0,C 180,E1 -12127.335,E2 -12127.335} C_VEL
LIN {X 0,Y 383.114,Z 739.722,A -85,B 0,C 180,E1 -12128.811,E2 -12128.811} C_VEL
LIN {X 0,Y 383.97,Z 745.669,A -85,B 0,C 180,E1 -12130.764,E2 -12130.764} C_VEL
LIN {X 0,Y 383.766,Z 752.822,A -85,B 0,C 180,E1 -12132.962,E2 -12132.962} C_VEL
LIN {X 0,Y 383.653,Z 755.548,A -85,B 0,C 180,E1 -12133.675,E2 -12133.675} C_VEL
LIN {X 0,Y 387.081,Z 774.492,A -85,B 0,C 180,E1 -12134.215,E2 -12134.215} C_VEL
LIN {X 0,Y 386.576,Z 830.891,A -85,B 0,C 180,E1 -12135.288,E2 -12135.288} C_VEL
LIN {X 0,Y 386.385,Z 839.896,A -85,B 0,C 180,E1 -12135.584,E2 -12135.584} C_VEL
LIN {X 0,Y 385.932,Z 849.445,A -85,B 0,C 180,E1 -12136.037,E2 -12136.037} C_VEL
LIN {X 0,Y 385.461,Z 859.455,A -85,B 0,C 180,E1 -12136.692,E2 -12136.692} C_VEL
LIN {X 0,Y 384.769,Z 869.838,A -85,B 0,C 180,E1 -12137.607,E2 -12137.607} C_VEL
LIN {X 0,Y 384.235,Z 877.965,A -85,B 0,C 180,E1 -12138.527,E2 -12138.527} C_VEL
LIN {X 0,Y 383.705,Z 884.67,A -85,B 0,C 180,E1 -12139.446,E2 -12139.446} C_VEL
LIN {X 0,Y 383.159,Z 891.018,A -85,B 0,C 180,E1 -12140.498,E2 -12140.498} C_VEL
LIN {X 0,Y 382.659,Z 897.46,A -85,B 0,C 180,E1 -12141.817,E2 -12141.817} C_VEL
LIN {X 0,Y 382.381,Z 902.019,A -85,B 0,C 180,E1 -12142.978,E2 -12142.978} C_VEL
LIN {X 0,Y 382.111,Z 905.867,A -85,B 0,C 180,E1 -12144.194,E2 -12144.194} C_VEL
LIN {X 0,Y 381.892,Z 908.525,A -85,B 0,C 180,E1 -12145.25,E2 -12145.25} C_VEL
LIN {X 0,Y 381.719,Z 911.433,A -85,B 0,C 180,E1 -12146.834,E2 -12146.834} C_VEL
LIN {X 0,Y 381.687,Z 912.703,A -85,B 0,C 180,E1 -12147.89,E2 -12147.89} C_VEL
LIN {X 0,Y 381.643,Z 913.506,A -85,B 0,C 180,E1 -12148.945,E2 -12148.945} C_VEL
LIN {X 0,Y 381.638,Z 913.811,A -85,B 0,C 180,E1 -12150,E2 -12150} C_VEL
LIN {X 0,Y 381.643,Z 913.535,A -85,B 0,C 180,E1 -12151.055,E2 -12151.055} C_VEL
LIN {X 0,Y 381.672,Z 912.792,A -85,B 0,C 180,E1 -12152.111,E2 -12152.111} C_VEL
LIN {X 0,Y 381.717,Z 911.581,A -85,B 0,C 180,E1 -12153.166,E2 -12153.166} C_VEL
LIN {X 0,Y 381.888,Z 908.735,A -85,B 0,C 180,E1 -12154.75,E2 -12154.75} C_VEL
LIN {X 0,Y 382.097,Z 906.144,A -85,B 0,C 180,E1 -12155.806,E2 -12155.806} C_VEL
LIN {X 0,Y 382.343,Z 902.537,A -85,B 0,C 180,E1 -12156.976,E2 -12156.976} C_VEL
LIN {X 0,Y 382.609,Z 897.891,A -85,B 0,C 180,E1 -12158.184,E2 -12158.184} C_VEL
LIN {X 0,Y 382.999,Z 892.949,A -85,B 0,C 180,E1 -12159.24,E2 -12159.24} C_VEL
LIN {X 0,Y 383.539,Z 886.981,A -85,B 0,C 180,E1 -12160.292,E2 -12160.292} C_VEL
LIN {X 0,Y 384.131,Z 879.716,A -85,B 0,C 180,E1 -12161.343,E2 -12161.343} C_VEL
LIN {X 0,Y 384.578,Z 873.177,A -85,B 0,C 180,E1 -12162.132,E2 -12162.132} C_VEL
LIN {X 0,Y 385.006,Z 866.752,A -85,B 0,C 180,E1 -12162.787,E2 -12162.787} C_VEL
LIN {X 0,Y 385.43,Z 860.053,A -85,B 0,C 180,E1 -12163.36,E2 -12163.36} C_VEL
LIN {X 0,Y 385.198,Z 854.762,A -85,B 0,C 180,E1 -12163.76,E2 -12163.76} C_VEL
LIN {X 0,Y 383.899,Z 849.534,A -85,B 0,C 180,E1 -12164.14,E2 -12164.14} C_VEL
LIN {X 0,Y 380.449,Z 837.991,A -85,B 0,C 180,E1 -12164.834,E2 -12164.834} C_VEL
LIN {X 0,Y 379.72,Z 831.346,A -85,B 0,C 180,E1 -12165.076,E2 -12165.076} C_VEL
LIN {X 0,Y 380.194,Z 774.536,A -85,B 0,C 180,E1 -12166.18,E2 -12166.18} C_VEL
LIN {X 0,Y 376.665,Z 755.373,A -85,B 0,C 180,E1 -12166.741,E2 -12166.741} C_VEL
LIN {X 0,Y 377.012,Z 747.966,A -85,B 0,C 180,E1 -12169.04,E2 -12169.04} C_VEL
LIN {X 0,Y 376.328,Z 742.067,A -85,B 0,C 180,E1 -12170.971,E2 -12170.971} C_VEL
LIN {X 0,Y 376.075,Z 740.541,A -85,B 0,C 180,E1 -12171.53,E2 -12171.53} C_VEL
LIN {X 0,Y 375.953,Z 740.468,A -85,B 0,C 180,E1 -12175.465,E2 -12175.465} C_VEL
LIN {X 0,Y 375.921,Z 740.47,A -85,B 0,C 180,E1 -12179.083,E2 -12179.083} C_VEL
LIN {X 0,Y 375.958,Z 740.454,A -85,B 0,C 180,E1 -12181.562,E2 -12181.562} C_VEL
LIN {X 0,Y 375.958,Z 740.466,A -85,B 0,C 180,E1 -12185.415,E2 -12185.415} C_VEL
LIN {X 0,Y 375.972,Z 740.444,A -85,B 0,C 180,E1 -12188.27,E2 -12188.27} C_VEL
LIN {X 0,Y 375.935,Z 740.466,A -85,B 0,C 180,E1 -12191.601,E2 -12191.601} C_VEL
LIN {X 0,Y 375.928,Z 740.454,A -85,B 0,C 180,E1 -12195.269,E2 -12195.269} C_VEL
LIN {X 0,Y 375.933,Z 740.43,A -85,B 0,C 180,E1 -12198.4,E2 -12198.4} C_VEL
LIN {X 0,Y 375.974,Z 740.459,A -85,B 0,C 180,E1 -12201.73,E2 -12201.73} C_VEL
LIN {X 0,Y 375.981,Z 740.455,A -85,B 0,C 180,E1 -12205.333,E2 -12205.333} C_VEL
LIN {X 0,Y 375.959,Z 740.459,A -85,B 0,C 180,E1 -12208.438,E2 -12208.438} C_VEL
LIN {X 0,Y 375.985,Z 740.457,A -85,B 0,C 180,E1 -12212.14,E2 -12212.14} C_VEL
LIN {X 0,Y 376.007,Z 740.443,A -85,B 0,C 180,E1 -12214.539,E2 -12214.539} C_VEL
LIN {X 0,Y 375.96,Z 740.463,A -85,B 0,C 180,E1 -12218.045,E2 -12218.045} C_VEL
LIN {X 0,Y 376.004,Z 740.446,A -85,B 0,C 180,E1 -12221.473,E2 -12221.473} C_VEL
LIN {X 0,Y 376.06,Z 740.443,A -85,B 0,C 180,E1 -12224.833,E2 -12224.833} C_VEL
LIN {X 0,Y 376.051,Z 740.451,A -85,B 0,C 180,E1 -12228.137,E2 -12228.137} C_VEL
LIN {X 0,Y 376.259,Z 740.405,A -85,B 0,C 180,E1 -12231.878,E2 -12231.878} C_VEL
LIN {X 0,Y 376.173,Z 740.428,A -85,B 0,C 180,E1 -12234.64,E2 -12234.64} C_VEL
LIN {X 0,Y 376.356,Z 740.415,A -85,B 0,C 180,E1 -12237.86,E2 -12237.86} C_VEL
LIN {X 0,Y 376.489,Z 740.389,A -85,B 0,C 180,E1 -12240,E2 -12240} C_VEL
LIN {X 0,Y 376.187,Z 740.416,A -85,B 0,C 180,E1 -12243.213,E2 -12243.213} C_VEL
LIN {X 0,Y 376.241,Z 740.428,A -85,B 0,C 180,E1 -12246.435,E2 -12246.435} C_VEL
LIN {X 0,Y 376.121,Z 740.44,A -85,B 0,C 180,E1 -12249.681,E2 -12249.681} C_VEL
LIN {X 0,Y 376.091,Z 740.435,A -85,B 0,C 180,E1 -12253.658,E2 -12253.658} C_VEL
LIN {X 0,Y 376.046,Z 740.456,A -85,B 0,C 180,E1 -12257.608,E2 -12257.608} C_VEL
LIN {X 0,Y 376.008,Z 740.441,A -85,B 0,C 180,E1 -12260.843,E2 -12260.843} C_VEL
LIN {X 0,Y 375.995,Z 740.462,A -85,B 0,C 180,E1 -12264.281,E2 -12264.281} C_VEL
LIN {X 0,Y 376.021,Z 740.454,A -85,B 0,C 180,E1 -12266.652,E2 -12266.652} C_VEL
LIN {X 0,Y 375.965,Z 740.456,A -85,B 0,C 180,E1 -12270.312,E2 -12270.312} C_VEL
LIN {X 0,Y 375.963,Z 740.467,A -85,B 0,C 180,E1 -12274.111,E2 -12274.111} C_VEL
LIN {X 0,Y 375.956,Z 740.445,A -85,B 0,C 180,E1 -12276.741,E2 -12276.741} C_VEL
LIN {X 0,Y 375.998,Z 740.416,A -85,B 0,C 180,E1 -12279.972,E2 -12279.972} C_VEL
LIN {X 0,Y 375.939,Z 740.464,A -85,B 0,C 180,E1 -12283.764,E2 -12283.764} C_VEL
LIN {X 0,Y 375.934,Z 740.46,A -85,B 0,C 180,E1 -12286.81,E2 -12286.81} C_VEL
LIN {X 0,Y 375.965,Z 740.461,A -85,B 0,C 180,E1 -12290.538,E2 -12290.538} C_VEL
LIN {X 0,Y 375.965,Z 740.457,A -85,B 0,C 180,E1 -12293.495,E2 -12293.495} C_VEL
LIN {X 0,Y 375.962,Z 740.465,A -85,B 0,C 180,E1 -12295.889,E2 -12295.889} C_VEL
LIN {X 0,Y 375.965,Z 740.443,A -85,B 0,C 180,E1 -12299.687,E2 -12299.687} C_VEL
LIN {X 0,Y 375.997,Z 740.459,A -85,B 0,C 180,E1 -12302.141,E2 -12302.141} C_VEL
LIN {X 0,Y 376.074,Z 740.58,A -85,B 0,C 180,E1 -12303.817,E2 -12303.817} C_VEL
LIN {X 0,Y 377.906,Z 750.721,A -85,B 0,C 180,E1 -12306.722,E2 -12306.722} C_VEL
LIN {X 0,Y 378.126,Z 753.978,A -85,B 0,C 180,E1 -12307.603,E2 -12307.603} C_VEL
LIN {X 0,Y 376.958,Z 768.974,A -85,B 0,C 180,E1 -12311.522,E2 -12311.522} C_VEL
LIN {X 0,Y 376.483,Z 775.82,A -85,B 0,C 180,E1 -12313.251,E2 -12313.251} C_VEL
LIN {X 0,Y 376.993,Z 779.567,A -85,B 0,C 180,E1 -12313.406,E2 -12313.406} C_VEL
LIN {X 0,Y 380.088,Z 802.373,A -85,B 0,C 180,E1 -12313.982,E2 -12313.982} C_VEL
LIN {X 0,Y 379.576,Z 852.412,A -85,B 0,C 180,E1 -12314.95,E2 -12314.95} C_VEL
LIN {X 0,Y 379.207,Z 862.162,A -85,B 0,C 180,E1 -12315.271,E2 -12315.271} C_VEL
LIN {X 0,Y 378.717,Z 872.207,A -85,B 0,C 180,E1 -12315.766,E2 -12315.766} C_VEL
LIN {X 0,Y 378.036,Z 883.618,A -85,B 0,C 180,E1 -12316.562,E2 -12316.562} C_VEL
LIN {X 0,Y 377.376,Z 892.207,A -85,B 0,C 180,E1 -12317.36,E2 -12317.36} C_VEL
LIN {X 0,Y 376.76,Z 900.291,A -85,B 0,C 180,E1 -12318.296,E2 -12318.296} C_VEL
LIN {X 0,Y 376.233,Z 906.971,A -85,B 0,C 180,E1 -12319.234,E2 -12319.234} C_VEL
LIN {X 0,Y 375.749,Z 913.314,A -85,B 0,C 180,E1 -12320.309,E2 -12320.309} C_VEL
LIN {X 0,Y 375.322,Z 918.584,A -85,B 0,C 180,E1 -12321.385,E2 -12321.385} C_VEL
LIN {X 0,Y 375.004,Z 922.981,A -85,B 0,C 180,E1 -12322.462,E2 -12322.462} C_VEL
LIN {X 0,Y 374.667,Z 928.345,A -85,B 0,C 180,E1 -12324.142,E2 -12324.142} C_VEL
LIN {X 0,Y 374.62,Z 931.978,A -85,B 0,C 180,E1 -12325.696,E2 -12325.696} C_VEL
LIN {X 0,Y 374.48,Z 933.728,A -85,B 0,C 180,E1 -12326.772,E2 -12326.772} C_VEL
LIN {X 0,Y 374.46,Z 934.983,A -85,B 0,C 180,E1 -12327.849,E2 -12327.849} C_VEL
LIN {X 0,Y 374.515,Z 935.766,A -85,B 0,C 180,E1 -12328.925,E2 -12328.925} C_VEL
LIN {X 0,Y 374.551,Z 936.063,A -85,B 0,C 180,E1 -12330,E2 -12330} C_VEL
LIN {X 0,Y 374.515,Z 935.764,A -85,B 0,C 180,E1 -12331.075,E2 -12331.075} C_VEL
LIN {X 0,Y 374.46,Z 934.976,A -85,B 0,C 180,E1 -12332.151,E2 -12332.151} C_VEL
LIN {X 0,Y 374.48,Z 933.716,A -85,B 0,C 180,E1 -12333.228,E2 -12333.228} C_VEL
LIN {X 0,Y 374.654,Z 930.804,A -85,B 0,C 180,E1 -12334.842,E2 -12334.842} C_VEL
LIN {X 0,Y 374.743,Z 927.089,A -85,B 0,C 180,E1 -12336.295,E2 -12336.295} C_VEL
LIN {X 0,Y 375.078,Z 921.989,A -85,B 0,C 180,E1 -12337.808,E2 -12337.808} C_VEL
LIN {X 0,Y 375.503,Z 916.111,A -85,B 0,C 180,E1 -12339.154,E2 -12339.154} C_VEL
LIN {X 0,Y 376.108,Z 908.635,A -85,B 0,C 180,E1 -12340.497,E2 -12340.497} C_VEL
LIN {X 0,Y 376.669,Z 901.264,A -85,B 0,C 180,E1 -12341.571,E2 -12341.571} C_VEL
LIN {X 0,Y 377.31,Z 893.373,A -85,B 0,C 180,E1 -12342.506,E2 -12342.506} C_VEL
LIN {X 0,Y 377.944,Z 885.036,A -85,B 0,C 180,E1 -12343.304,E2 -12343.304} C_VEL
LIN {X 0,Y 378.608,Z 874.389,A -85,B 0,C 180,E1 -12344.101,E2 -12344.101} C_VEL
LIN {X 0,Y 379.134,Z 862.802,A -85,B 0,C 180,E1 -12344.698,E2 -12344.698} C_VEL
LIN {X 0,Y 379.558,Z 853.103,A -85,B 0,C 180,E1 -12345.024,E2 -12345.024} C_VEL
LIN {X 0,Y 379.991,Z 801.138,A -85,B 0,C 180,E1 -12346.037,E2 -12346.037} C_VEL
LIN {X 0,Y 376.483,Z 776.15,A -85,B 0,C 180,E1 -12346.704,E2 -12346.704} C_VEL
LIN {X 0,Y 376.607,Z 773.217,A -85,B 0,C 180,E1 -12347.372,E2 -12347.372} C_VEL
LIN {X 0,Y 377.575,Z 760.398,A -85,B 0,C 180,E1 -12350.711,E2 -12350.711} C_VEL
LIN {X 0,Y 378.168,Z 752.867,A -85,B 0,C 180,E1 -12352.683,E2 -12352.683} C_VEL
LIN {X 0,Y 376.522,Z 743.099,A -85,B 0,C 180,E1 -12355.424,E2 -12355.424} C_VEL
LIN {X 0,Y 376.059,Z 740.48,A -85,B 0,C 180,E1 -12356.244,E2 -12356.244} C_VEL
LIN {X 0,Y 375.971,Z 740.459,A -85,B 0,C 180,E1 -12359.079,E2 -12359.079} C_VEL
LIN {X 0,Y 375.951,Z 740.464,A -85,B 0,C 180,E1 -12362.828,E2 -12362.828} C_VEL
LIN {X 0,Y 375.959,Z 740.459,A -85,B 0,C 180,E1 -12365.415,E2 -12365.415} C_VEL
LIN {X 0,Y 375.977,Z 740.462,A -85,B 0,C 180,E1 -12368.271,E2 -12368.271} C_VEL
LIN {X 0,Y 375.935,Z 740.452,A -85,B 0,C 180,E1 -12371.601,E2 -12371.601} C_VEL
LIN {X 0,Y 375.928,Z 740.471,A -85,B 0,C 180,E1 -12375.269,E2 -12375.269} C_VEL
LIN {X 0,Y 375.961,Z 740.444,A -85,B 0,C 180,E1 -12378.395,E2 -12378.395} C_VEL
LIN {X 0,Y 375.978,Z 740.423,A -85,B 0,C 180,E1 -12381.729,E2 -12381.729} C_VEL
LIN {X 0,Y 375.981,Z 740.458,A -85,B 0,C 180,E1 -12385.333,E2 -12385.333} C_VEL
LIN {X 0,Y 375.959,Z 740.46,A -85,B 0,C 180,E1 -12388.438,E2 -12388.438} C_VEL
LIN {X 0,Y 375.984,Z 740.458,A -85,B 0,C 180,E1 -12392.141,E2 -12392.141} C_VEL
LIN {X 0,Y 376.007,Z 740.458,A -85,B 0,C 180,E1 -12394.539,E2 -12394.539} C_VEL
LIN {X 0,Y 375.968,Z 740.449,A -85,B 0,C 180,E1 -12398.046,E2 -12398.046} C_VEL
LIN {X 0,Y 376.031,Z 740.451,A -85,B 0,C 180,E1 -12401.474,E2 -12401.474} C_VEL
LIN {X 0,Y 376.06,Z 740.446,A -85,B 0,C 180,E1 -12404.833,E2 -12404.833} C_VEL
LIN {X 0,Y 376.051,Z 740.435,A -85,B 0,C 180,E1 -12408.137,E2 -12408.137} C_VEL
LIN {X 0,Y 376.22,Z 740.431,A -85,B 0,C 180,E1 -12411.919,E2 -12411.919} C_VEL
LIN {X 0,Y 376.172,Z 740.433,A -85,B 0,C 180,E1 -12414.64,E2 -12414.64} C_VEL
LIN {X 0,Y 376.354,Z 740.392,A -85,B 0,C 180,E1 -12417.86,E2 -12417.86} C_VEL
LIN {X 0,Y 376.491,Z 740.389,A -85,B 0,C 180,E1 -12420,E2 -12420} C_VEL
LIN {X 0,Y 376.192,Z 740.434,A -85,B 0,C 180,E1 -12423.213,E2 -12423.213} C_VEL
LIN {X 0,Y 376.238,Z 740.413,A -85,B 0,C 180,E1 -12426.568,E2 -12426.568} C_VEL
LIN {X 0,Y 376.207,Z 740.416,A -85,B 0,C 180,E1 -12428.595,E2 -12428.595} C_VEL
LIN {X 0,Y 376.051,Z 740.451,A -85,B 0,C 180,E1 -12431.863,E2 -12431.863} C_VEL
LIN {X 0,Y 376.06,Z 740.443,A -85,B 0,C 180,E1 -12435.167,E2 -12435.167} C_VEL
LIN {X 0,Y 376.004,Z 740.445,A -85,B 0,C 180,E1 -12438.527,E2 -12438.527} C_VEL
LIN {X 0,Y 375.958,Z 740.463,A -85,B 0,C 180,E1 -12441.955,E2 -12441.955} C_VEL
LIN {X 0,Y 376.007,Z 740.443,A -85,B 0,C 180,E1 -12445.461,E2 -12445.461} C_VEL
LIN {X 0,Y 375.962,Z 740.466,A -85,B 0,C 180,E1 -12449.08,E2 -12449.08} C_VEL
LIN {X 0,Y 375.95,Z 740.459,A -85,B 0,C 180,E1 -12452.829,E2 -12452.829} C_VEL
LIN {X 0,Y 375.958,Z 740.465,A -85,B 0,C 180,E1 -12455.416,E2 -12455.416} C_VEL
LIN {X 0,Y 375.974,Z 740.459,A -85,B 0,C 180,E1 -12458.27,E2 -12458.27} C_VEL
LIN {X 0,Y 375.933,Z 740.431,A -85,B 0,C 180,E1 -12461.6,E2 -12461.6} C_VEL
LIN {X 0,Y 375.928,Z 740.457,A -85,B 0,C 180,E1 -12465.269,E2 -12465.269} C_VEL
LIN {X 0,Y 375.935,Z 740.466,A -85,B 0,C 180,E1 -12468.399,E2 -12468.399} C_VEL
LIN {X 0,Y 375.973,Z 740.444,A -85,B 0,C 180,E1 -12471.73,E2 -12471.73} C_VEL
LIN {X 0,Y 375.981,Z 740.467,A -85,B 0,C 180,E1 -12475.333,E2 -12475.333} C_VEL
LIN {X 0,Y 375.958,Z 740.453,A -85,B 0,C 180,E1 -12478.438,E2 -12478.438} C_VEL
LIN {X 0,Y 375.936,Z 740.468,A -85,B 0,C 180,E1 -12482.136,E2 -12482.136} C_VEL
